LIN {X 0,Y 305.104,Z 484.661,A -85,B 0,C 180,E1 7191.33,E2 7191.33} C_VEL
LIN {X 0,Y 307.303,Z 489.456,A -85,B 0,C 180,E1 7188.457,E2 7188.457} C_VEL
LIN {X 0,Y 307.394,Z 489.963,A -85,B 0,C 180,E1 7188.319,E2 7188.319} C_VEL
LIN {X 0,Y 295.914,Z 597.326,A -85,B 0,C 180,E1 7186.379,E2 7186.379} C_VEL
LIN {X 0,Y 291.472,Z 621.219,A -85,B 0,C 180,E1 7185.834,E2 7185.834} C_VEL
LIN {X 0,Y 286.108,Z 641.71,A -85,B 0,C 180,E1 7185.236,E2 7185.236} C_VEL
LIN {X 0,Y 278.769,Z 663.649,A -85,B 0,C 180,E1 7184.366,E2 7184.366} C_VEL
LIN {X 0,Y 271.258,Z 681.916,A -85,B 0,C 180,E1 7183.403,E2 7183.403} C_VEL
LIN {X 0,Y 262.549,Z 700.2,A -85,B 0,C 180,E1 7182.184,E2 7182.184} C_VEL
LIN {X 0,Y 251.426,Z 720.077,A -85,B 0,C 180,E1 7180.47,E2 7180.47} C_VEL
LIN {X 0,Y 241.401,Z 735.774,A -85,B 0,C 180,E1 7178.733,E2 7178.733} C_VEL
LIN {X 0,Y 229.63,Z 752.334,A -85,B 0,C 180,E1 7176.424,E2 7176.424} C_VEL
LIN {X 0,Y 216.754,Z 768.298,A -85,B 0,C 180,E1 7173.492,E2 7173.492} C_VEL
LIN {X 0,Y 205.612,Z 780.95,A -85,B 0,C 180,E1 7170.508,E2 7170.508} C_VEL
LIN {X 0,Y 192.249,Z 794.919,A -85,B 0,C 180,E1 7166.187,E2 7166.187} C_VEL
LIN {X 0,Y 189.925,Z 797.18,A -85,B 0,C 180,E1 7165.331,E2 7165.331} C_VEL
LIN {X 0,Y 185.106,Z 801.348,A -85,B 0,C 180,E1 7163.939,E2 7163.939} C_VEL
LIN {X 0,Y 170.53,Z 810.999,A -85,B 0,C 180,E1 7160.73,E2 7160.73} C_VEL
LIN {X 0,Y 165.908,Z 814.382,A -85,B 0,C 180,E1 7158.968,E2 7158.968} C_VEL
LIN {X 0,Y 154.577,Z 824.022,A -85,B 0,C 180,E1 7151.776,E2 7151.776} C_VEL
LIN {X 0,Y 146.89,Z 830.6,A -85,B 0,C 180,E1 7144.873,E2 7144.873} C_VEL
LIN {X 0,Y 140.749,Z 836.382,A -85,B 0,C 180,E1 7136.481,E2 7136.481} C_VEL
LIN {X 0,Y 137.18,Z 840.393,A -85,B 0,C 180,E1 7127.387,E2 7127.387} C_VEL
LIN {X 0,Y 136.118,Z 842.389,A -85,B 0,C 180,E1 7120.154,E2 7120.154} C_VEL
LIN {X 0,Y 136.006,Z 843.295,A -85,B 0,C 180,E1 7113.794,E2 7113.794} C_VEL
LIN {X 0,Y 136.026,Z 843.438,A -85,B 0,C 180,E1 7108.315,E2 7108.315} C_VEL
LIN {X 0,Y 136.046,Z 842.73,A -85,B 0,C 180,E1 7101.548,E2 7101.548} C_VEL
LIN {X 0,Y 136.809,Z 840.957,A -85,B 0,C 180,E1 7094.312,E2 7094.312} C_VEL
LIN {X 0,Y 139.161,Z 837.954,A -85,B 0,C 180,E1 7086.724,E2 7086.724} C_VEL
LIN {X 0,Y 143.968,Z 833.277,A -85,B 0,C 180,E1 7078.61,E2 7078.61} C_VEL
LIN {X 0,Y 151.933,Z 826.255,A -85,B 0,C 180,E1 7070.333,E2 7070.333} C_VEL
LIN {X 0,Y 160.416,Z 819.053,A -85,B 0,C 180,E1 7064.212,E2 7064.212} C_VEL
LIN {X 0,Y 171.771,Z 809.365,A -85,B 0,C 180,E1 7058.098,E2 7058.098} C_VEL
LIN {X 0,Y 183.827,Z 798.354,A -85,B 0,C 180,E1 7053.112,E2 7053.112} C_VEL
LIN {X 0,Y 195.767,Z 786.783,A -85,B 0,C 180,E1 7049.151,E2 7049.151} C_VEL
LIN {X 0,Y 210.081,Z 771.62,A -85,B 0,C 180,E1 7045.276,E2 7045.276} C_VEL
LIN {X 0,Y 221.987,Z 757.619,A -85,B 0,C 180,E1 7042.583,E2 7042.583} C_VEL
LIN {X 0,Y 234.35,Z 741.577,A -85,B 0,C 180,E1 7040.181,E2 7040.181} C_VEL
LIN {X 0,Y 246.233,Z 723.952,A -85,B 0,C 180,E1 7038.166,E2 7038.166} C_VEL
LIN {X 0,Y 256.353,Z 706.973,A -85,B 0,C 180,E1 7036.645,E2 7036.645} C_VEL
LIN {X 0,Y 266.872,Z 686.5,A -85,B 0,C 180,E1 7035.225,E2 7035.225} C_VEL
LIN {X 0,Y 274.893,Z 667.932,A -85,B 0,C 180,E1 7034.233,E2 7034.233} C_VEL
LIN {X 0,Y 282.326,Z 647.454,A -85,B 0,C 180,E1 7033.391,E2 7033.391} C_VEL
LIN {X 0,Y 288.635,Z 625.044,A -85,B 0,C 180,E1 7032.726,E2 7032.726} C_VEL
LIN {X 0,Y 293.049,Z 603.912,A -85,B 0,C 180,E1 7032.239,E2 7032.239} C_VEL
LIN {X 0,Y 296.866,Z 573.803,A -85,B 0,C 180,E1 7031.673,E2 7031.673} C_VEL
LIN {X 0,Y 305.233,Z 495.411,A -85,B 0,C 180,E1 7030.284,E2 7030.284} C_VEL
LIN {X 0,Y 303.319,Z 491.087,A -85,B 0,C 180,E1 7027.386,E2 7027.386} C_VEL
LIN {X 0,Y 302.008,Z 487.906,A -85,B 0,C 180,E1 7024.367,E2 7024.367} C_VEL
LIN {X 0,Y 301.205,Z 486.572,A -85,B 0,C 180,E1 7019.81,E2 7019.81} C_VEL
LIN {X 0,Y 302.134,Z 488.028,A -85,B 0,C 180,E1 7014.874,E2 7014.874} C_VEL
LIN {X 0,Y 303.893,Z 492.391,A -85,B 0,C 180,E1 7011.2,E2 7011.2} C_VEL
LIN {X 0,Y 307.885,Z 499.46,A -85,B 0,C 180,E1 7006.478,E2 7006.478} C_VEL
LIN {X 0,Y 312.909,Z 504.765,A -85,B 0,C 180,E1 7002.617,E2 7002.617} C_VEL
LIN {X 0,Y 316.473,Z 507.473,A -85,B 0,C 180,E1 7000.434,E2 7000.434} C_VEL
LIN {X 0,Y 321.483,Z 511.596,A -85,B 0,C 180,E1 6997.315,E2 6997.315} C_VEL
LIN {X 0,Y 325.724,Z 514.379,A -85,B 0,C 180,E1 6994.353,E2 6994.353} C_VEL
LIN {X 0,Y 327.911,Z 515.873,A -85,B 0,C 180,E1 6992.684,E2 6992.684} C_VEL
LIN {X 0,Y 331.07,Z 519.079,A -85,B 0,C 180,E1 6989.912,E2 6989.912} C_VEL
LIN {X 0,Y 334.513,Z 521.924,A -85,B 0,C 180,E1 6986.43,E2 6986.43} C_VEL
LIN {X 0,Y 336.136,Z 523.16,A -85,B 0,C 180,E1 6984.756,E2 6984.756} C_VEL
LIN {X 0,Y 338.877,Z 526.467,A -85,B 0,C 180,E1 6981.703,E2 6981.703} C_VEL
LIN {X 0,Y 342.275,Z 529.188,A -85,B 0,C 180,E1 6978.013,E2 6978.013} C_VEL
LIN {X 0,Y 344.04,Z 530.411,A -85,B 0,C 180,E1 6976.006,E2 6976.006} C_VEL
LIN {X 0,Y 347.045,Z 534.052,A -85,B 0,C 180,E1 6972.232,E2 6972.232} C_VEL
LIN {X 0,Y 349.83,Z 536.292,A -85,B 0,C 180,E1 6968.715,E2 6968.715} C_VEL
LIN {X 0,Y 352.358,Z 537.818,A -85,B 0,C 180,E1 6965.37,E2 6965.37} C_VEL
LIN {X 0,Y 354.546,Z 540.837,A -85,B 0,C 180,E1 6961.913,E2 6961.913} C_VEL
LIN {X 0,Y 356.813,Z 542.935,A -85,B 0,C 180,E1 6958.265,E2 6958.265} C_VEL
LIN {X 0,Y 358.894,Z 544.236,A -85,B 0,C 180,E1 6954.525,E2 6954.525} C_VEL
LIN {X 0,Y 360.791,Z 545.097,A -85,B 0,C 180,E1 6950.776,E2 6950.776} C_VEL
LIN {X 0,Y 361.998,Z 546.95,A -85,B 0,C 180,E1 6947.521,E2 6947.521} C_VEL
LIN {X 0,Y 363.22,Z 548.56,A -85,B 0,C 180,E1 6943.856,E2 6943.856} C_VEL
LIN {X 0,Y 364.051,Z 549.551,A -85,B 0,C 180,E1 6940.443,E2 6940.443} C_VEL
LIN {X 0,Y 364.784,Z 550.154,A -85,B 0,C 180,E1 6936.768,E2 6936.768} C_VEL
LIN {X 0,Y 365.112,Z 550.448,A -85,B 0,C 180,E1 6933.454,E2 6933.454} C_VEL
LIN {X 0,Y 365.309,Z 550.567,A -85,B 0,C 180,E1 6929.843,E2 6929.843} C_VEL
LIN {X 0,Y 365.099,Z 550.448,A -85,B 0,C 180,E1 6926.389,E2 6926.389} C_VEL
LIN {X 0,Y 364.734,Z 550.083,A -85,B 0,C 180,E1 6922.756,E2 6922.756} C_VEL
LIN {X 0,Y 363.978,Z 549.471,A -85,B 0,C 180,E1 6919.234,E2 6919.234} C_VEL
LIN {X 0,Y 363.085,Z 548.4,A -85,B 0,C 180,E1 6915.651,E2 6915.651} C_VEL
LIN {X 0,Y 361.936,Z 546.859,A -85,B 0,C 180,E1 6912.31,E2 6912.31} C_VEL
LIN {X 0,Y 360.733,Z 545.031,A -85,B 0,C 180,E1 6909.051,E2 6909.051} C_VEL
LIN {X 0,Y 358.895,Z 544.236,A -85,B 0,C 180,E1 6905.475,E2 6905.475} C_VEL
LIN {X 0,Y 356.813,Z 542.935,A -85,B 0,C 180,E1 6901.735,E2 6901.735} C_VEL
LIN {X 0,Y 354.546,Z 540.837,A -85,B 0,C 180,E1 6898.087,E2 6898.087} C_VEL
LIN {X 0,Y 352.358,Z 537.819,A -85,B 0,C 180,E1 6894.63,E2 6894.63} C_VEL
LIN {X 0,Y 349.461,Z 536.056,A -85,B 0,C 180,E1 6890.838,E2 6890.838} C_VEL
LIN {X 0,Y 346.883,Z 533.875,A -85,B 0,C 180,E1 6887.552,E2 6887.552} C_VEL
LIN {X 0,Y 343.927,Z 530.256,A -85,B 0,C 180,E1 6883.866,E2 6883.866} C_VEL
LIN {X 0,Y 340.638,Z 528.014,A -85,B 0,C 180,E1 6880.222,E2 6880.222} C_VEL
LIN {X 0,Y 337.257,Z 524.656,A -85,B 0,C 180,E1 6876.471,E2 6876.471} C_VEL
LIN {X 0,Y 335.469,Z 522.476,A -85,B 0,C 180,E1 6874.492,E2 6874.492} C_VEL
LIN {X 0,Y 331.8,Z 519.751,A -85,B 0,C 180,E1 6870.816,E2 6870.816} C_VEL
LIN {X 0,Y 328.541,Z 516.579,A -85,B 0,C 180,E1 6867.849,E2 6867.849} C_VEL
LIN {X 0,Y 326.725,Z 514.885,A -85,B 0,C 180,E1 6866.342,E2 6866.342} C_VEL
LIN {X 0,Y 322.538,Z 512.398,A -85,B 0,C 180,E1 6863.427,E2 6863.427} C_VEL
LIN {X 0,Y 317.626,Z 508.513,A -85,B 0,C 180,E1 6860.259,E2 6860.259} C_VEL
LIN {X 0,Y 314.164,Z 505.643,A -85,B 0,C 180,E1 6858.173,E2 6858.173} C_VEL
LIN {X 0,Y 308.694,Z 500.604,A -85,B 0,C 180,E1 6854.251,E2 6854.251} C_VEL
LIN {X 0,Y 305.593,Z 495.836,A -85,B 0,C 180,E1 6851.13,E2 6851.13} C_VEL
LIN {X 0,Y 303.288,Z 491.023,A -85,B 0,C 180,E1 6847.768,E2 6847.768} C_VEL
LIN {X 0,Y 301.987,Z 487.887,A -85,B 0,C 180,E1 6844.748,E2 6844.748} C_VEL
LIN {X 0,Y 301.205,Z 486.57,A -85,B 0,C 180,E1 6840.19,E2 6840.19} C_VEL
LIN {X 0,Y 302.119,Z 488.008,A -85,B 0,C 180,E1 6835.349,E2 6835.349} C_VEL
LIN {X 0,Y 303.866,Z 492.356,A -85,B 0,C 180,E1 6831.675,E2 6831.675} C_VEL
LIN {X 0,Y 305.234,Z 495.59,A -85,B 0,C 180,E1 6829.692,E2 6829.692} C_VEL
LIN {X 0,Y 294.112,Z 597.19,A -85,B 0,C 180,E1 6827.898,E2 6827.898} C_VEL
LIN {X 0,Y 289.582,Z 621.099,A -85,B 0,C 180,E1 6827.372,E2 6827.372} C_VEL
LIN {X 0,Y 284.203,Z 641.339,A -85,B 0,C 180,E1 6826.808,E2 6826.808} C_VEL
LIN {X 0,Y 276.75,Z 663.292,A -85,B 0,C 180,E1 6825.979,E2 6825.979} C_VEL
LIN {X 0,Y 268.823,Z 682.187,A -85,B 0,C 180,E1 6825.024,E2 6825.024} C_VEL
LIN {X 0,Y 259.301,Z 701.676,A -85,B 0,C 180,E1 6823.762,E2 6823.762} C_VEL
LIN {X 0,Y 248.577,Z 720.215,A -85,B 0,C 180,E1 6822.2,E2 6822.2} C_VEL
LIN {X 0,Y 238.137,Z 736.139,A -85,B 0,C 180,E1 6820.489,E2 6820.489} C_VEL
LIN {X 0,Y 225.247,Z 753.642,A -85,B 0,C 180,E1 6818.081,E2 6818.081} C_VEL
LIN {X 0,Y 212.424,Z 768.939,A -85,B 0,C 180,E1 6815.286,E2 6815.286} C_VEL
LIN {X 0,Y 200.185,Z 782.301,A -85,B 0,C 180,E1 6812.133,E2 6812.133} C_VEL
LIN {X 0,Y 186.553,Z 795.792,A -85,B 0,C 180,E1 6807.865,E2 6807.865} C_VEL
LIN {X 0,Y 175.348,Z 806.096,A -85,B 0,C 180,E1 6803.512,E2 6803.512} C_VEL
LIN {X 0,Y 165.908,Z 814.382,A -85,B 0,C 180,E1 6798.968,E2 6798.968} C_VEL
LIN {X 0,Y 161.388,Z 817.688,A -85,B 0,C 180,E1 6797.08,E2 6797.08} C_VEL
LIN {X 0,Y 147.59,Z 825.211,A -85,B 0,C 180,E1 6792.401,E2 6792.401} C_VEL
LIN {X 0,Y 143.546,Z 827.744,A -85,B 0,C 180,E1 6789.986,E2 6789.986} C_VEL
LIN {X 0,Y 135.713,Z 834.039,A -85,B 0,C 180,E1 6781.539,E2 6781.539} C_VEL
LIN {X 0,Y 131.259,Z 838.095,A -85,B 0,C 180,E1 6773.81,E2 6773.81} C_VEL
LIN {X 0,Y 128.634,Z 841.269,A -85,B 0,C 180,E1 6764.862,E2 6764.862} C_VEL
LIN {X 0,Y 128.003,Z 842.929,A -85,B 0,C 180,E1 6755.828,E2 6755.828} C_VEL
LIN {X 0,Y 128.039,Z 843.245,A -85,B 0,C 180,E1 6749.105,E2 6749.105} C_VEL
LIN {X 0,Y 128.035,Z 842.65,A -85,B 0,C 180,E1 6741.92,E2 6741.92} C_VEL
LIN {X 0,Y 128.976,Z 840.706,A -85,B 0,C 180,E1 6733.332,E2 6733.332} C_VEL
LIN {X 0,Y 131.655,Z 837.701,A -85,B 0,C 180,E1 6725.311,E2 6725.311} C_VEL
LIN {X 0,Y 137.315,Z 832.769,A -85,B 0,C 180,E1 6716.401,E2 6716.401} C_VEL
LIN {X 0,Y 146.11,Z 825.628,A -85,B 0,C 180,E1 6707.886,E2 6707.886} C_VEL
LIN {X 0,Y 155.297,Z 818.363,A -85,B 0,C 180,E1 6701.683,E2 6701.683} C_VEL
LIN {X 0,Y 167.939,Z 808.113,A -85,B 0,C 180,E1 6695.35,E2 6695.35} C_VEL
LIN {X 0,Y 180.145,Z 797.46,A -85,B 0,C 180,E1 6690.653,E2 6690.653} C_VEL
LIN {X 0,Y 192.636,Z 785.812,A -85,B 0,C 180,E1 6686.782,E2 6686.782} C_VEL
LIN {X 0,Y 207.505,Z 770.473,A -85,B 0,C 180,E1 6683.029,E2 6683.029} C_VEL
LIN {X 0,Y 219.801,Z 756.374,A -85,B 0,C 180,E1 6680.438,E2 6680.438} C_VEL
LIN {X 0,Y 232.949,Z 739.582,A -85,B 0,C 180,E1 6678.068,E2 6678.068} C_VEL
LIN {X 0,Y 244.696,Z 722.328,A -85,B 0,C 180,E1 6676.217,E2 6676.217} C_VEL
LIN {X 0,Y 255.803,Z 703.856,A -85,B 0,C 180,E1 6674.676,E2 6674.676} C_VEL
LIN {X 0,Y 265.724,Z 684.378,A -85,B 0,C 180,E1 6673.431,E2 6673.431} C_VEL
LIN {X 0,Y 273.48,Z 666.555,A -85,B 0,C 180,E1 6672.542,E2 6672.542} C_VEL
LIN {X 0,Y 281.084,Z 645.615,A -85,B 0,C 180,E1 6671.741,E2 6671.741} C_VEL
LIN {X 0,Y 287.297,Z 623.474,A -85,B 0,C 180,E1 6671.13,E2 6671.13} C_VEL
LIN {X 0,Y 291.807,Z 601.687,A -85,B 0,C 180,E1 6670.655,E2 6670.655} C_VEL
LIN {X 0,Y 295.891,Z 568.531,A -85,B 0,C 180,E1 6670.06,E2 6670.06} C_VEL
LIN {X 0,Y 303.217,Z 501.505,A -85,B 0,C 180,E1 6668.916,E2 6668.916} C_VEL
LIN {X 0,Y 302.021,Z 498.596,A -85,B 0,C 180,E1 6666.845,E2 6666.845} C_VEL
LIN {X 0,Y 300.963,Z 495.798,A -85,B 0,C 180,E1 6664.191,E2 6664.191} C_VEL
LIN {X 0,Y 300.23,Z 494.512,A -85,B 0,C 180,E1 6659.809,E2 6659.809} C_VEL
LIN {X 0,Y 301.08,Z 495.958,A -85,B 0,C 180,E1 6655.047,E2 6655.047} C_VEL
LIN {X 0,Y 302.72,Z 500.238,A -85,B 0,C 180,E1 6651.452,E2 6651.452} C_VEL
LIN {X 0,Y 306.511,Z 507.154,A -85,B 0,C 180,E1 6646.8,E2 6646.8} C_VEL
LIN {X 0,Y 311.554,Z 512.565,A -85,B 0,C 180,E1 6642.827,E2 6642.827} C_VEL
LIN {X 0,Y 315.236,Z 515.434,A -85,B 0,C 180,E1 6640.547,E2 6640.547} C_VEL
LIN {X 0,Y 320.279,Z 519.511,A -85,B 0,C 180,E1 6637.419,E2 6637.419} C_VEL
LIN {X 0,Y 324.569,Z 522.278,A -85,B 0,C 180,E1 6634.451,E2 6634.451} C_VEL
LIN {X 0,Y 326.675,Z 523.725,A -85,B 0,C 180,E1 6632.868,E2 6632.868} C_VEL
LIN {X 0,Y 329.974,Z 527.007,A -85,B 0,C 180,E1 6630.002,E2 6630.002} C_VEL
LIN {X 0,Y 333.437,Z 529.838,A -85,B 0,C 180,E1 6626.513,E2 6626.513} C_VEL
LIN {X 0,Y 335.057,Z 531.131,A -85,B 0,C 180,E1 6624.849,E2 6624.849} C_VEL
LIN {X 0,Y 337.987,Z 534.563,A -85,B 0,C 180,E1 6621.594,E2 6621.594} C_VEL
LIN {X 0,Y 341.397,Z 537.221,A -85,B 0,C 180,E1 6617.881,E2 6617.881} C_VEL
LIN {X 0,Y 342.997,Z 538.414,A -85,B 0,C 180,E1 6616.055,E2 6616.055} C_VEL
LIN {X 0,Y 346.014,Z 541.999,A -85,B 0,C 180,E1 6612.29,E2 6612.29} C_VEL
LIN {X 0,Y 348.889,Z 544.276,A -85,B 0,C 180,E1 6608.663,E2 6608.663} C_VEL
LIN {X 0,Y 351.365,Z 545.841,A -85,B 0,C 180,E1 6605.373,E2 6605.373} C_VEL
LIN {X 0,Y 353.555,Z 548.808,A -85,B 0,C 180,E1 6601.926,E2 6601.926} C_VEL
LIN {X 0,Y 355.893,Z 550.929,A -85,B 0,C 180,E1 6598.162,E2 6598.162} C_VEL
LIN {X 0,Y 357.98,Z 552.213,A -85,B 0,C 180,E1 6594.416,E2 6594.416} C_VEL
LIN {X 0,Y 359.918,Z 553.152,A -85,B 0,C 180,E1 6590.489,E2 6590.489} C_VEL
LIN {X 0,Y 361.2,Z 555.135,A -85,B 0,C 180,E1 6587.063,E2 6587.063} C_VEL
LIN {X 0,Y 362.335,Z 556.681,A -85,B 0,C 180,E1 6583.403,E2 6583.403} C_VEL
LIN {X 0,Y 363.152,Z 557.557,A -85,B 0,C 180,E1 6580.149,E2 6580.149} C_VEL
LIN {X 0,Y 363.837,Z 558.169,A -85,B 0,C 180,E1 6576.311,E2 6576.311} C_VEL
LIN {X 0,Y 364.171,Z 558.392,A -85,B 0,C 180,E1 6573.148,E2 6573.148} C_VEL
LIN {X 0,Y 364.271,Z 558.474,A -85,B 0,C 180,E1 6569.214,E2 6569.214} C_VEL
LIN {X 0,Y 364.104,Z 558.382,A -85,B 0,C 180,E1 6566.064,E2 6566.064} C_VEL
LIN {X 0,Y 363.626,Z 557.966,A -85,B 0,C 180,E1 6562.257,E2 6562.257} C_VEL
LIN {X 0,Y 362.964,Z 557.365,A -85,B 0,C 180,E1 6559.043,E2 6559.043} C_VEL
LIN {X 0,Y 361.931,Z 556.198,A -85,B 0,C 180,E1 6555.216,E2 6555.216} C_VEL
LIN {X 0,Y 360.821,Z 554.591,A -85,B 0,C 180,E1 6551.892,E2 6551.892} C_VEL
LIN {X 0,Y 359.66,Z 552.924,A -85,B 0,C 180,E1 6548.814,E2 6548.814} C_VEL
LIN {X 0,Y 357.774,Z 552.107,A -85,B 0,C 180,E1 6545.217,E2 6545.217} C_VEL
LIN {X 0,Y 355.654,Z 550.764,A -85,B 0,C 180,E1 6541.451,E2 6541.451} C_VEL
LIN {X 0,Y 353.372,Z 548.597,A -85,B 0,C 180,E1 6537.78,E2 6537.78} C_VEL
LIN {X 0,Y 350.934,Z 545.355,A -85,B 0,C 180,E1 6534.013,E2 6534.013} C_VEL
LIN {X 0,Y 348.262,Z 543.866,A -85,B 0,C 180,E1 6530.561,E2 6530.561} C_VEL
LIN {X 0,Y 345.413,Z 541.344,A -85,B 0,C 180,E1 6526.912,E2 6526.912} C_VEL
LIN {X 0,Y 342.236,Z 537.7,A -85,B 0,C 180,E1 6523.083,E2 6523.083} C_VEL
LIN {X 0,Y 338.9,Z 535.355,A -85,B 0,C 180,E1 6519.369,E2 6519.369} C_VEL
LIN {X 0,Y 335.707,Z 532.044,A -85,B 0,C 180,E1 6515.895,E2 6515.895} C_VEL
LIN {X 0,Y 334.207,Z 530.288,A -85,B 0,C 180,E1 6514.225,E2 6514.225} C_VEL
LIN {X 0,Y 330.693,Z 527.675,A -85,B 0,C 180,E1 6510.729,E2 6510.729} C_VEL
LIN {X 0,Y 327.403,Z 524.538,A -85,B 0,C 180,E1 6507.757,E2 6507.757} C_VEL
LIN {X 0,Y 325.563,Z 522.782,A -85,B 0,C 180,E1 6506.247,E2 6506.247} C_VEL
LIN {X 0,Y 321.293,Z 520.261,A -85,B 0,C 180,E1 6503.28,E2 6503.28} C_VEL
LIN {X 0,Y 316.092,Z 516.207,A -85,B 0,C 180,E1 6499.976,E2 6499.976} C_VEL
LIN {X 0,Y 312.652,Z 513.348,A -85,B 0,C 180,E1 6497.879,E2 6497.879} C_VEL
LIN {X 0,Y 307.197,Z 508.156,A -85,B 0,C 180,E1 6493.841,E2 6493.841} C_VEL
LIN {X 0,Y 304.217,Z 503.402,A -85,B 0,C 180,E1 6490.702,E2 6490.702} C_VEL
LIN {X 0,Y 302.093,Z 498.728,A -85,B 0,C 180,E1 6487.416,E2 6487.416} C_VEL
LIN {X 0,Y 300.944,Z 495.778,A -85,B 0,C 180,E1 6484.573,E2 6484.573} C_VEL
LIN {X 0,Y 300.23,Z 494.511,A -85,B 0,C 180,E1 6480.191,E2 6480.191} C_VEL
LIN {X 0,Y 301.069,Z 495.911,A -85,B 0,C 180,E1 6475.524,E2 6475.524} C_VEL
LIN {X 0,Y 302.693,Z 500.201,A -85,B 0,C 180,E1 6471.93,E2 6471.93} C_VEL
LIN {X 0,Y 303.193,Z 501.752,A -85,B 0,C 180,E1 6471.075,E2 6471.075} C_VEL
LIN {X 0,Y 292.52,Z 597.054,A -85,B 0,C 180,E1 6469.435,E2 6469.435} C_VEL
LIN {X 0,Y 287.904,Z 620.979,A -85,B 0,C 180,E1 6468.929,E2 6468.929} C_VEL
LIN {X 0,Y 282.244,Z 641.883,A -85,B 0,C 180,E1 6468.373,E2 6468.373} C_VEL
LIN {X 0,Y 274.4,Z 664.292,A -85,B 0,C 180,E1 6467.557,E2 6467.557} C_VEL
LIN {X 0,Y 266.55,Z 682.583,A -85,B 0,C 180,E1 6466.668,E2 6466.668} C_VEL
LIN {X 0,Y 256.582,Z 702.448,A -85,B 0,C 180,E1 6465.425,E2 6465.425} C_VEL
LIN {X 0,Y 245.576,Z 720.953,A -85,B 0,C 180,E1 6463.913,E2 6463.913} C_VEL
LIN {X 0,Y 235.102,Z 736.504,A -85,B 0,C 180,E1 6462.291,E2 6462.291} C_VEL
LIN {X 0,Y 222.007,Z 753.757,A -85,B 0,C 180,E1 6459.984,E2 6459.984} C_VEL
LIN {X 0,Y 209.119,Z 768.686,A -85,B 0,C 180,E1 6457.334,E2 6457.334} C_VEL
LIN {X 0,Y 196.465,Z 782.047,A -85,B 0,C 180,E1 6454.26,E2 6454.26} C_VEL
LIN {X 0,Y 182.205,Z 795.61,A -85,B 0,C 180,E1 6450.042,E2 6450.042} C_VEL
LIN {X 0,Y 170.54,Z 805.849,A -85,B 0,C 180,E1 6445.748,E2 6445.748} C_VEL
LIN {X 0,Y 158.134,Z 816.181,A -85,B 0,C 180,E1 6439.911,E2 6439.911} C_VEL
LIN {X 0,Y 147.526,Z 824.512,A -85,B 0,C 180,E1 6433.197,E2 6433.197} C_VEL
LIN {X 0,Y 143.546,Z 827.744,A -85,B 0,C 180,E1 6429.986,E2 6429.986} C_VEL
LIN {X 0,Y 139.719,Z 830.079,A -85,B 0,C 180,E1 6427.42,E2 6427.42} C_VEL
LIN {X 0,Y 127.339,Z 835.519,A -85,B 0,C 180,E1 6420.361,E2 6420.361} C_VEL
LIN {X 0,Y 124.923,Z 836.877,A -85,B 0,C 180,E1 6417.603,E2 6417.603} C_VEL
LIN {X 0,Y 121.418,Z 840.172,A -85,B 0,C 180,E1 6408.732,E2 6408.732} C_VEL
LIN {X 0,Y 120.14,Z 842.06,A -85,B 0,C 180,E1 6400.55,E2 6400.55} C_VEL
LIN {X 0,Y 120.011,Z 842.828,A -85,B 0,C 180,E1 6393.822,E2 6393.822} C_VEL
LIN {X 0,Y 120.03,Z 842.942,A -85,B 0,C 180,E1 6388.091,E2 6388.091} C_VEL
LIN {X 0,Y 120.067,Z 842.316,A -85,B 0,C 180,E1 6380.896,E2 6380.896} C_VEL
LIN {X 0,Y 121.181,Z 840.455,A -85,B 0,C 180,E1 6372.225,E2 6372.225} C_VEL
LIN {X 0,Y 124.234,Z 837.448,A -85,B 0,C 180,E1 6363.728,E2 6363.728} C_VEL
LIN {X 0,Y 130.508,Z 832.515,A -85,B 0,C 180,E1 6354.392,E2 6354.392} C_VEL
LIN {X 0,Y 140.071,Z 825.373,A -85,B 0,C 180,E1 6345.611,E2 6345.611} C_VEL
LIN {X 0,Y 149.906,Z 818.107,A -85,B 0,C 180,E1 6339.314,E2 6339.314} C_VEL
LIN {X 0,Y 163.283,Z 807.854,A -85,B 0,C 180,E1 6332.977,E2 6332.977} C_VEL
LIN {X 0,Y 176.068,Z 797.206,A -85,B 0,C 180,E1 6328.335,E2 6328.335} C_VEL
LIN {X 0,Y 189.848,Z 784.84,A -85,B 0,C 180,E1 6324.342,E2 6324.342} C_VEL
LIN {X 0,Y 204.427,Z 770.22,A -85,B 0,C 180,E1 6320.907,E2 6320.907} C_VEL
LIN {X 0,Y 217.073,Z 756.123,A -85,B 0,C 180,E1 6318.409,E2 6318.409} C_VEL
LIN {X 0,Y 230.806,Z 738.968,A -85,B 0,C 180,E1 6316.096,E2 6316.096} C_VEL
LIN {X 0,Y 242.547,Z 722.078,A -85,B 0,C 180,E1 6314.369,E2 6314.369} C_VEL
LIN {X 0,Y 253.869,Z 703.601,A -85,B 0,C 180,E1 6312.904,E2 6312.904} C_VEL
LIN {X 0,Y 263.962,Z 684.13,A -85,B 0,C 180,E1 6311.723,E2 6311.723} C_VEL
LIN {X 0,Y 271.843,Z 666.311,A -85,B 0,C 180,E1 6310.882,E2 6310.882} C_VEL
LIN {X 0,Y 279.582,Z 645.287,A -85,B 0,C 180,E1 6310.124,E2 6310.124} C_VEL
LIN {X 0,Y 285.87,Z 623.176,A -85,B 0,C 180,E1 6309.549,E2 6309.549} C_VEL
LIN {X 0,Y 290.461,Z 601.249,A -85,B 0,C 180,E1 6309.093,E2 6309.093} C_VEL
LIN {X 0,Y 294.664,Z 567.644,A -85,B 0,C 180,E1 6308.511,E2 6308.511} C_VEL
LIN {X 0,Y 301.352,Z 507.516,A -85,B 0,C 180,E1 6307.483,E2 6307.483} C_VEL
LIN {X 0,Y 299.922,Z 503.689,A -85,B 0,C 180,E1 6304.014,E2 6304.014} C_VEL
LIN {X 0,Y 299.256,Z 502.456,A -85,B 0,C 180,E1 6299.617,E2 6299.617} C_VEL
LIN {X 0,Y 300.055,Z 504.002,A -85,B 0,C 180,E1 6295.126,E2 6295.126} C_VEL
LIN {X 0,Y 301.502,Z 507.934,A -85,B 0,C 180,E1 6291.802,E2 6291.802} C_VEL
LIN {X 0,Y 305.522,Z 515.426,A -85,B 0,C 180,E1 6286.757,E2 6286.757} C_VEL
LIN {X 0,Y 310.604,Z 520.663,A -85,B 0,C 180,E1 6282.773,E2 6282.773} C_VEL
LIN {X 0,Y 314.002,Z 523.39,A -85,B 0,C 180,E1 6280.661,E2 6280.661} C_VEL
LIN {X 0,Y 319.064,Z 527.423,A -85,B 0,C 180,E1 6277.523,E2 6277.523} C_VEL
LIN {X 0,Y 323.505,Z 530.225,A -85,B 0,C 180,E1 6274.483,E2 6274.483} C_VEL
LIN {X 0,Y 325.554,Z 531.707,A -85,B 0,C 180,E1 6272.954,E2 6272.954} C_VEL
LIN {X 0,Y 329.054,Z 535.105,A -85,B 0,C 180,E1 6269.91,E2 6269.91} C_VEL
LIN {X 0,Y 332.551,Z 537.87,A -85,B 0,C 180,E1 6266.412,E2 6266.412} C_VEL
LIN {X 0,Y 333.917,Z 539.012,A -85,B 0,C 180,E1 6265.011,E2 6265.011} C_VEL
LIN {X 0,Y 336.926,Z 542.498,A -85,B 0,C 180,E1 6261.668,E2 6261.668} C_VEL
LIN {X 0,Y 340.35,Z 545.143,A -85,B 0,C 180,E1 6257.948,E2 6257.948} C_VEL
LIN {X 0,Y 341.819,Z 546.232,A -85,B 0,C 180,E1 6256.26,E2 6256.26} C_VEL
LIN {X 0,Y 344.863,Z 549.826,A -85,B 0,C 180,E1 6252.494,E2 6252.494} C_VEL
LIN {X 0,Y 347.591,Z 552.036,A -85,B 0,C 180,E1 6249.044,E2 6249.044} C_VEL
LIN {X 0,Y 350.271,Z 553.685,A -85,B 0,C 180,E1 6245.557,E2 6245.557} C_VEL
LIN {X 0,Y 352.525,Z 556.735,A -85,B 0,C 180,E1 6242,E2 6242} C_VEL
LIN {X 0,Y 354.74,Z 558.767,A -85,B 0,C 180,E1 6238.431,E2 6238.431} C_VEL
LIN {X 0,Y 356.857,Z 560.083,A -85,B 0,C 180,E1 6234.675,E2 6234.675} C_VEL
LIN {X 0,Y 358.797,Z 560.954,A -85,B 0,C 180,E1 6230.897,E2 6230.897} C_VEL
LIN {X 0,Y 360.065,Z 562.906,A -85,B 0,C 180,E1 6227.451,E2 6227.451} C_VEL
LIN {X 0,Y 361.287,Z 564.507,A -85,B 0,C 180,E1 6223.739,E2 6223.739} C_VEL
LIN {X 0,Y 362.126,Z 565.462,A -85,B 0,C 180,E1 6220.339,E2 6220.339} C_VEL
LIN {X 0,Y 362.838,Z 566.06,A -85,B 0,C 180,E1 6216.646,E2 6216.646} C_VEL
LIN {X 0,Y 363.177,Z 566.33,A -85,B 0,C 180,E1 6213.314,E2 6213.314} C_VEL
LIN {X 0,Y 363.339,Z 566.44,A -85,B 0,C 180,E1 6209.685,E2 6209.685} C_VEL
LIN {X 0,Y 363.148,Z 566.328,A -85,B 0,C 180,E1 6206.369,E2 6206.369} C_VEL
LIN {X 0,Y 362.799,Z 565.974,A -85,B 0,C 180,E1 6202.812,E2 6202.812} C_VEL
LIN {X 0,Y 362.049,Z 565.388,A -85,B 0,C 180,E1 6199.337,E2 6199.337} C_VEL
LIN {X 0,Y 361.148,Z 564.309,A -85,B 0,C 180,E1 6195.694,E2 6195.694} C_VEL
LIN {X 0,Y 359.943,Z 562.732,A -85,B 0,C 180,E1 6192.209,E2 6192.209} C_VEL
LIN {X 0,Y 358.738,Z 560.892,A -85,B 0,C 180,E1 6188.928,E2 6188.928} C_VEL
LIN {X 0,Y 356.801,Z 560.053,A -85,B 0,C 180,E1 6185.222,E2 6185.222} C_VEL
LIN {X 0,Y 354.731,Z 558.761,A -85,B 0,C 180,E1 6181.554,E2 6181.554} C_VEL
LIN {X 0,Y 352.505,Z 556.713,A -85,B 0,C 180,E1 6177.968,E2 6177.968} C_VEL
LIN {X 0,Y 350.233,Z 553.626,A -85,B 0,C 180,E1 6174.383,E2 6174.383} C_VEL
LIN {X 0,Y 347.238,Z 551.797,A -85,B 0,C 180,E1 6170.506,E2 6170.506} C_VEL
LIN {X 0,Y 344.487,Z 549.408,A -85,B 0,C 180,E1 6166.995,E2 6166.995} C_VEL
LIN {X 0,Y 341.578,Z 545.894,A -85,B 0,C 180,E1 6163.455,E2 6163.455} C_VEL
LIN {X 0,Y 338.296,Z 543.659,A -85,B 0,C 180,E1 6159.787,E2 6159.787} C_VEL
LIN {X 0,Y 334.925,Z 540.369,A -85,B 0,C 180,E1 6156.129,E2 6156.129} C_VEL
LIN {X 0,Y 333.026,Z 538.142,A -85,B 0,C 180,E1 6154.042,E2 6154.042} C_VEL
LIN {X 0,Y 329.588,Z 535.598,A -85,B 0,C 180,E1 6150.641,E2 6150.641} C_VEL
LIN {X 0,Y 326.281,Z 532.509,A -85,B 0,C 180,E1 6147.676,E2 6147.676} C_VEL
LIN {X 0,Y 324.15,Z 530.557,A -85,B 0,C 180,E1 6145.977,E2 6145.977} C_VEL
LIN {X 0,Y 319.865,Z 527.99,A -85,B 0,C 180,E1 6143,E2 6143} C_VEL
LIN {X 0,Y 314.566,Z 523.9,A -85,B 0,C 180,E1 6139.69,E2 6139.69} C_VEL
LIN {X 0,Y 311.15,Z 521.052,A -85,B 0,C 180,E1 6137.581,E2 6137.581} C_VEL
LIN {X 0,Y 305.814,Z 515.847,A -85,B 0,C 180,E1 6133.519,E2 6133.519} C_VEL
LIN {X 0,Y 302.786,Z 510.841,A -85,B 0,C 180,E1 6130.176,E2 6130.176} C_VEL
LIN {X 0,Y 300.911,Z 506.432,A -85,B 0,C 180,E1 6127.062,E2 6127.062} C_VEL
LIN {X 0,Y 299.903,Z 503.669,A -85,B 0,C 180,E1 6124.398,E2 6124.398} C_VEL
LIN {X 0,Y 299.258,Z 502.448,A -85,B 0,C 180,E1 6120,E2 6120} C_VEL
LIN {X 0,Y 300.07,Z 504.069,A -85,B 0,C 180,E1 6115.509,E2 6115.509} C_VEL
LIN {X 0,Y 301.365,Z 507.617,A -85,B 0,C 180,E1 6112.482,E2 6112.482} C_VEL
LIN {X 0,Y 291.139,Z 596.913,A -85,B 0,C 180,E1 6110.987,E2 6110.987} C_VEL
LIN {X 0,Y 286.47,Z 620.74,A -85,B 0,C 180,E1 6110.506,E2 6110.506} C_VEL
LIN {X 0,Y 280.499,Z 642.424,A -85,B 0,C 180,E1 6109.959,E2 6109.959} C_VEL
LIN {X 0,Y 272.776,Z 664.047,A -85,B 0,C 180,E1 6109.211,E2 6109.211} C_VEL
LIN {X 0,Y 264.884,Z 682.158,A -85,B 0,C 180,E1 6108.38,E2 6108.38} C_VEL
LIN {X 0,Y 255.239,Z 701.166,A -85,B 0,C 180,E1 6107.263,E2 6107.263} C_VEL
LIN {X 0,Y 243.895,Z 720.017,A -85,B 0,C 180,E1 6105.816,E2 6105.816} C_VEL
LIN {X 0,Y 232.747,Z 736.253,A -85,B 0,C 180,E1 6104.208,E2 6104.208} C_VEL
LIN {X 0,Y 218.791,Z 754.135,A -85,B 0,C 180,E1 6101.9,E2 6101.9} C_VEL
LIN {X 0,Y 206.09,Z 768.433,A -85,B 0,C 180,E1 6099.444,E2 6099.444} C_VEL
LIN {X 0,Y 192.23,Z 782.596,A -85,B 0,C 180,E1 6096.265,E2 6096.265} C_VEL
LIN {X 0,Y 177.518,Z 795.956,A -85,B 0,C 180,E1 6092.128,E2 6092.128} C_VEL
LIN {X 0,Y 164.647,Z 806.722,A -85,B 0,C 180,E1 6087.574,E2 6087.574} C_VEL
LIN {X 0,Y 150.5,Z 817.672,A -85,B 0,C 180,E1 6081.012,E2 6081.012} C_VEL
LIN {X 0,Y 140.27,Z 825.225,A -85,B 0,C 180,E1 6074.536,E2 6074.536} C_VEL
LIN {X 0,Y 130.679,Z 832.393,A -85,B 0,C 180,E1 6065.803,E2 6065.803} C_VEL
LIN {X 0,Y 124.923,Z 836.877,A -85,B 0,C 180,E1 6057.603,E2 6057.603} C_VEL
LIN {X 0,Y 122.308,Z 838.359,A -85,B 0,C 180,E1 6054.279,E2 6054.279} C_VEL
LIN {X 0,Y 115.553,Z 840.537,A -85,B 0,C 180,E1 6047.836,E2 6047.836} C_VEL
LIN {X 0,Y 112.498,Z 841.535,A -85,B 0,C 180,E1 6043.035,E2 6043.035} C_VEL
LIN {X 0,Y 112.215,Z 841.758,A -85,B 0,C 180,E1 6041.623,E2 6041.623} C_VEL
LIN {X 0,Y 112.012,Z 842.58,A -85,B 0,C 180,E1 6034.095,E2 6034.095} C_VEL
LIN {X 0,Y 112.031,Z 842.694,A -85,B 0,C 180,E1 6027.954,E2 6027.954} C_VEL
LIN {X 0,Y 112.092,Z 842.066,A -85,B 0,C 180,E1 6020.243,E2 6020.243} C_VEL
LIN {X 0,Y 113.433,Z 840.203,A -85,B 0,C 180,E1 6010.966,E2 6010.966} C_VEL
LIN {X 0,Y 117.174,Z 836.998,A -85,B 0,C 180,E1 6001.456,E2 6001.456} C_VEL
LIN {X 0,Y 124.697,Z 831.701,A -85,B 0,C 180,E1 5991.288,E2 5991.288} C_VEL
LIN {X 0,Y 134.813,Z 824.746,A -85,B 0,C 180,E1 5982.758,E2 5982.758} C_VEL
LIN {X 0,Y 146.326,Z 816.802,A -85,B 0,C 180,E1 5975.99,E2 5975.99} C_VEL
LIN {X 0,Y 161.075,Z 805.899,A -85,B 0,C 180,E1 5969.656,E2 5969.656} C_VEL
LIN {X 0,Y 174.621,Z 795.031,A -85,B 0,C 180,E1 5965.222,E2 5965.222} C_VEL
LIN {X 0,Y 189.885,Z 781.54,A -85,B 0,C 180,E1 5961.254,E2 5961.254} C_VEL
LIN {X 0,Y 203.348,Z 768.18,A -85,B 0,C 180,E1 5958.387,E2 5958.387} C_VEL
LIN {X 0,Y 217.266,Z 752.88,A -85,B 0,C 180,E1 5955.889,E2 5955.889} C_VEL
LIN {X 0,Y 231.214,Z 735.242,A -85,B 0,C 180,E1 5953.759,E2 5953.759} C_VEL
LIN {X 0,Y 242.488,Z 719.08,A -85,B 0,C 180,E1 5952.258,E2 5952.258} C_VEL
LIN {X 0,Y 254.501,Z 699.214,A -85,B 0,C 180,E1 5950.843,E2 5950.843} C_VEL
LIN {X 0,Y 263.843,Z 680.923,A -85,B 0,C 180,E1 5949.847,E2 5949.847} C_VEL
LIN {X 0,Y 272.33,Z 661.528,A -85,B 0,C 180,E1 5949.03,E2 5949.03} C_VEL
LIN {X 0,Y 279.923,Z 639.837,A -85,B 0,C 180,E1 5948.354,E2 5948.354} C_VEL
LIN {X 0,Y 285.774,Z 618.42,A -85,B 0,C 180,E1 5947.86,E2 5947.86} C_VEL
LIN {X 0,Y 290.222,Z 594.937,A -85,B 0,C 180,E1 5947.415,E2 5947.415} C_VEL
LIN {X 0,Y 299.655,Z 513.953,A -85,B 0,C 180,E1 5946.086,E2 5946.086} C_VEL
LIN {X 0,Y 298.822,Z 511.51,A -85,B 0,C 180,E1 5943.645,E2 5943.645} C_VEL
LIN {X 0,Y 298.281,Z 510.396,A -85,B 0,C 180,E1 5939.616,E2 5939.616} C_VEL
LIN {X 0,Y 298.982,Z 511.809,A -85,B 0,C 180,E1 5935.396,E2 5935.396} C_VEL
LIN {X 0,Y 300.294,Z 515.629,A -85,B 0,C 180,E1 5932.154,E2 5932.154} C_VEL
LIN {X 0,Y 304.345,Z 523.399,A -85,B 0,C 180,E1 5926.898,E2 5926.898} C_VEL
LIN {X 0,Y 309.655,Z 528.756,A -85,B 0,C 180,E1 5922.719,E2 5922.719} C_VEL
LIN {X 0,Y 316.598,Z 534.427,A -85,B 0,C 180,E1 5918.413,E2 5918.413} C_VEL
LIN {X 0,Y 321.006,Z 537.381,A -85,B 0,C 180,E1 5915.527,E2 5915.527} C_VEL
LIN {X 0,Y 324.042,Z 539.301,A -85,B 0,C 180,E1 5913.324,E2 5913.324} C_VEL
LIN {X 0,Y 327.751,Z 542.86,A -85,B 0,C 180,E1 5910.181,E2 5910.181} C_VEL
LIN {X 0,Y 331.236,Z 545.634,A -85,B 0,C 180,E1 5906.733,E2 5906.733} C_VEL
LIN {X 0,Y 332.759,Z 546.877,A -85,B 0,C 180,E1 5905.187,E2 5905.187} C_VEL
LIN {X 0,Y 335.866,Z 550.433,A -85,B 0,C 180,E1 5901.742,E2 5901.742} C_VEL
LIN {X 0,Y 339.302,Z 553.065,A -85,B 0,C 180,E1 5898.016,E2 5898.016} C_VEL
LIN {X 0,Y 340.79,Z 554.246,A -85,B 0,C 180,E1 5896.295,E2 5896.295} C_VEL
LIN {X 0,Y 343.775,Z 557.715,A -85,B 0,C 180,E1 5892.622,E2 5892.622} C_VEL
LIN {X 0,Y 346.565,Z 559.966,A -85,B 0,C 180,E1 5889.097,E2 5889.097} C_VEL
LIN {X 0,Y 349.248,Z 561.661,A -85,B 0,C 180,E1 5885.604,E2 5885.604} C_VEL
LIN {X 0,Y 351.515,Z 564.683,A -85,B 0,C 180,E1 5882.045,E2 5882.045} C_VEL
LIN {X 0,Y 353.809,Z 566.755,A -85,B 0,C 180,E1 5878.343,E2 5878.343} C_VEL
LIN {X 0,Y 355.983,Z 568.081,A -85,B 0,C 180,E1 5874.491,E2 5874.491} C_VEL
LIN {X 0,Y 357.921,Z 569.009,A -85,B 0,C 180,E1 5870.608,E2 5870.608} C_VEL
LIN {X 0,Y 359.2,Z 571.004,A -85,B 0,C 180,E1 5867.161,E2 5867.161} C_VEL
LIN {X 0,Y 360.401,Z 572.616,A -85,B 0,C 180,E1 5863.312,E2 5863.312} C_VEL
LIN {X 0,Y 361.233,Z 573.457,A -85,B 0,C 180,E1 5860.042,E2 5860.042} C_VEL
LIN {X 0,Y 361.883,Z 574.048,A -85,B 0,C 180,E1 5856.345,E2 5856.345} C_VEL
LIN {X 0,Y 362.22,Z 574.273,A -85,B 0,C 180,E1 5853.165,E2 5853.165} C_VEL
LIN {X 0,Y 362.333,Z 574.362,A -85,B 0,C 180,E1 5849.368,E2 5849.368} C_VEL
LIN {X 0,Y 362.161,Z 574.266,A -85,B 0,C 180,E1 5846.201,E2 5846.201} C_VEL
LIN {X 0,Y 361.747,Z 573.874,A -85,B 0,C 180,E1 5842.536,E2 5842.536} C_VEL
LIN {X 0,Y 361.031,Z 573.285,A -85,B 0,C 180,E1 5839.145,E2 5839.145} C_VEL
LIN {X 0,Y 360.032,Z 572.147,A -85,B 0,C 180,E1 5835.362,E2 5835.362} C_VEL
LIN {X 0,Y 358.892,Z 570.578,A -85,B 0,C 180,E1 5831.987,E2 5831.987} C_VEL
LIN {X 0,Y 357.729,Z 568.821,A -85,B 0,C 180,E1 5828.866,E2 5828.866} C_VEL
LIN {X 0,Y 355.805,Z 567.988,A -85,B 0,C 180,E1 5825.185,E2 5825.185} C_VEL
LIN {X 0,Y 353.692,Z 566.673,A -85,B 0,C 180,E1 5821.462,E2 5821.462} C_VEL
LIN {X 0,Y 351.332,Z 564.472,A -85,B 0,C 180,E1 5817.655,E2 5817.655} C_VEL
LIN {X 0,Y 348.697,Z 561.133,A -85,B 0,C 180,E1 5813.682,E2 5813.682} C_VEL
LIN {X 0,Y 345.948,Z 559.532,A -85,B 0,C 180,E1 5810.088,E2 5810.088} C_VEL
LIN {X 0,Y 342.899,Z 556.827,A -85,B 0,C 180,E1 5806.314,E2 5806.314} C_VEL
LIN {X 0,Y 340.014,Z 553.47,A -85,B 0,C 180,E1 5802.788,E2 5802.788} C_VEL
LIN {X 0,Y 336.413,Z 550.911,A -85,B 0,C 180,E1 5798.838,E2 5798.838} C_VEL
LIN {X 0,Y 333.252,Z 547.572,A -85,B 0,C 180,E1 5795.384,E2 5795.384} C_VEL
LIN {X 0,Y 331.86,Z 546.008,A -85,B 0,C 180,E1 5793.875,E2 5793.875} C_VEL
LIN {X 0,Y 328.46,Z 543.494,A -85,B 0,C 180,E1 5790.52,E2 5790.52} C_VEL
LIN {X 0,Y 324.921,Z 540.226,A -85,B 0,C 180,E1 5787.39,E2 5787.39} C_VEL
LIN {X 0,Y 322.744,Z 538.33,A -85,B 0,C 180,E1 5785.704,E2 5785.704} C_VEL
LIN {X 0,Y 318.395,Z 535.713,A -85,B 0,C 180,E1 5782.722,E2 5782.722} C_VEL
LIN {X 0,Y 313.189,Z 531.718,A -85,B 0,C 180,E1 5779.488,E2 5779.488} C_VEL
LIN {X 0,Y 309.386,Z 528.562,A -85,B 0,C 180,E1 5777.103,E2 5777.103} C_VEL
LIN {X 0,Y 304.157,Z 523.118,A -85,B 0,C 180,E1 5772.917,E2 5772.917} C_VEL
LIN {X 0,Y 301.449,Z 518.403,A -85,B 0,C 180,E1 5769.739,E2 5769.739} C_VEL
LIN {X 0,Y 299.739,Z 514.135,A -85,B 0,C 180,E1 5766.705,E2 5766.705} C_VEL
LIN {X 0,Y 298.866,Z 511.559,A -85,B 0,C 180,E1 5764.221,E2 5764.221} C_VEL
LIN {X 0,Y 298.283,Z 510.389,A -85,B 0,C 180,E1 5760,E2 5760} C_VEL
LIN {X 0,Y 298.995,Z 511.874,A -85,B 0,C 180,E1 5755.781,E2 5755.781} C_VEL
LIN {X 0,Y 299.649,Z 514.096,A -85,B 0,C 180,E1 5753.894,E2 5753.894} C_VEL
LIN {X 0,Y 289.96,Z 596.862,A -85,B 0,C 180,E1 5752.552,E2 5752.552} C_VEL
LIN {X 0,Y 285.225,Z 620.62,A -85,B 0,C 180,E1 5752.095,E2 5752.095} C_VEL
LIN {X 0,Y 279.209,Z 642.184,A -85,B 0,C 180,E1 5751.584,E2 5751.584} C_VEL
LIN {X 0,Y 271.382,Z 663.803,A -85,B 0,C 180,E1 5750.884,E2 5750.884} C_VEL
LIN {X 0,Y 263.374,Z 681.909,A -85,B 0,C 180,E1 5750.105,E2 5750.105} C_VEL
LIN {X 0,Y 253.109,Z 701.722,A -85,B 0,C 180,E1 5748.999,E2 5748.999} C_VEL
LIN {X 0,Y 241.571,Z 720.455,A -85,B 0,C 180,E1 5747.627,E2 5747.627} C_VEL
LIN {X 0,Y 230.207,Z 736.618,A -85,B 0,C 180,E1 5746.096,E2 5746.096} C_VEL
LIN {X 0,Y 215.714,Z 754.64,A -85,B 0,C 180,E1 5743.853,E2 5743.853} C_VEL
LIN {X 0,Y 202.493,Z 769.073,A -85,B 0,C 180,E1 5741.445,E2 5741.445} C_VEL
LIN {X 0,Y 187.417,Z 783.845,A -85,B 0,C 180,E1 5738.164,E2 5738.164} C_VEL
LIN {X 0,Y 173.066,Z 796.312,A -85,B 0,C 180,E1 5734.321,E2 5734.321} C_VEL
LIN {X 0,Y 159.638,Z 807.035,A -85,B 0,C 180,E1 5729.804,E2 5729.804} C_VEL
LIN {X 0,Y 145.424,Z 817.416,A -85,B 0,C 180,E1 5723.553,E2 5723.553} C_VEL
LIN {X 0,Y 134.813,Z 824.746,A -85,B 0,C 180,E1 5717.242,E2 5717.242} C_VEL
LIN {X 0,Y 124.697,Z 831.701,A -85,B 0,C 180,E1 5708.712,E2 5708.712} C_VEL
LIN {X 0,Y 117.117,Z 837.041,A -85,B 0,C 180,E1 5698.438,E2 5698.438} C_VEL
LIN {X 0,Y 113.433,Z 840.203,A -85,B 0,C 180,E1 5689.034,E2 5689.034} C_VEL
LIN {X 0,Y 112.215,Z 841.758,A -85,B 0,C 180,E1 5681.623,E2 5681.623} C_VEL
LIN {X 0,Y 111.118,Z 842.322,A -85,B 0,C 180,E1 5677.979,E2 5677.979} C_VEL
LIN {X 0,Y 108.09,Z 842.534,A -85,B 0,C 180,E1 5672.959,E2 5672.959} C_VEL
LIN {X 0,Y 104.182,Z 842.31,A -85,B 0,C 180,E1 5664.912,E2 5664.912} C_VEL
LIN {X 0,Y 104.02,Z 842.193,A -85,B 0,C 180,E1 5663.035,E2 5663.035} C_VEL
LIN {X 0,Y 105.19,Z 840.516,A -85,B 0,C 180,E1 5651.72,E2 5651.72} C_VEL
LIN {X 0,Y 109.154,Z 837.337,A -85,B 0,C 180,E1 5640.957,E2 5640.957} C_VEL
LIN {X 0,Y 116.154,Z 832.77,A -85,B 0,C 180,E1 5631.07,E2 5631.07} C_VEL
LIN {X 0,Y 127.779,Z 825.49,A -85,B 0,C 180,E1 5621.094,E2 5621.094} C_VEL
LIN {X 0,Y 139.319,Z 818.029,A -85,B 0,C 180,E1 5614.381,E2 5614.381} C_VEL
LIN {X 0,Y 153.398,Z 808.441,A -85,B 0,C 180,E1 5608.368,E2 5608.368} C_VEL
LIN {X 0,Y 168.044,Z 797.339,A -85,B 0,C 180,E1 5603.613,E2 5603.613} C_VEL
LIN {X 0,Y 182.972,Z 784.924,A -85,B 0,C 180,E1 5599.804,E2 5599.804} C_VEL
LIN {X 0,Y 199.151,Z 769.714,A -85,B 0,C 180,E1 5596.483,E2 5596.483} C_VEL
LIN {X 0,Y 212.951,Z 755.083,A -85,B 0,C 180,E1 5594.132,E2 5594.132} C_VEL
LIN {X 0,Y 227.534,Z 737.504,A -85,B 0,C 180,E1 5592.029,E2 5592.029} C_VEL
LIN {X 0,Y 239.492,Z 720.893,A -85,B 0,C 180,E1 5590.529,E2 5590.529} C_VEL
LIN {X 0,Y 251.215,Z 702.278,A -85,B 0,C 180,E1 5589.236,E2 5589.236} C_VEL
LIN {X 0,Y 261.63,Z 682.648,A -85,B 0,C 180,E1 5588.199,E2 5588.199} C_VEL
LIN {X 0,Y 269.995,Z 664.094,A -85,B 0,C 180,E1 5587.447,E2 5587.447} C_VEL
LIN {X 0,Y 278.146,Z 641.944,A -85,B 0,C 180,E1 5586.777,E2 5586.777} C_VEL
LIN {X 0,Y 284.382,Z 619.783,A -85,B 0,C 180,E1 5586.29,E2 5586.29} C_VEL
LIN {X 0,Y 289.192,Z 595.532,A -85,B 0,C 180,E1 5585.85,E2 5585.85} C_VEL
LIN {X 0,Y 298.119,Z 520.506,A -85,B 0,C 180,E1 5584.66,E2 5584.66} C_VEL
LIN {X 0,Y 297.79,Z 519.399,A -85,B 0,C 180,E1 5583.465,E2 5583.465} C_VEL
LIN {X 0,Y 297.311,Z 518.337,A -85,B 0,C 180,E1 5579.422,E2 5579.422} C_VEL
LIN {X 0,Y 297.96,Z 519.845,A -85,B 0,C 180,E1 5575.477,E2 5575.477} C_VEL
LIN {X 0,Y 299.099,Z 523.324,A -85,B 0,C 180,E1 5572.509,E2 5572.509} C_VEL
LIN {X 0,Y 305.801,Z 534.476,A -85,B 0,C 180,E1 5564.74,E2 5564.74} C_VEL
LIN {X 0,Y 310.788,Z 538.638,A -85,B 0,C 180,E1 5561.331,E2 5561.331} C_VEL
LIN {X 0,Y 316.37,Z 543.05,A -85,B 0,C 180,E1 5557.908,E2 5557.908} C_VEL
LIN {X 0,Y 321.107,Z 545.974,A -85,B 0,C 180,E1 5554.749,E2 5554.749} C_VEL
LIN {X 0,Y 323.098,Z 547.5,A -85,B 0,C 180,E1 5553.239,E2 5553.239} C_VEL
LIN {X 0,Y 326.841,Z 550.954,A -85,B 0,C 180,E1 5550.09,E2 5550.09} C_VEL
LIN {X 0,Y 330.321,Z 553.649,A -85,B 0,C 180,E1 5546.658,E2 5546.658} C_VEL
LIN {X 0,Y 331.68,Z 554.858,A -85,B 0,C 180,E1 5545.268,E2 5545.268} C_VEL
LIN {X 0,Y 334.875,Z 558.429,A -85,B 0,C 180,E1 5541.742,E2 5541.742} C_VEL
LIN {X 0,Y 338.254,Z 560.987,A -85,B 0,C 180,E1 5538.084,E2 5538.084} C_VEL
LIN {X 0,Y 339.652,Z 562.11,A -85,B 0,C 180,E1 5536.462,E2 5536.462} C_VEL
LIN {X 0,Y 342.624,Z 565.534,A -85,B 0,C 180,E1 5532.838,E2 5532.838} C_VEL
LIN {X 0,Y 345.39,Z 567.797,A -85,B 0,C 180,E1 5529.343,E2 5529.343} C_VEL
LIN {X 0,Y 348.139,Z 569.533,A -85,B 0,C 180,E1 5525.755,E2 5525.755} C_VEL
LIN {X 0,Y 350.505,Z 572.63,A -85,B 0,C 180,E1 5522.089,E2 5522.089} C_VEL
LIN {X 0,Y 352.769,Z 574.669,A -85,B 0,C 180,E1 5518.434,E2 5518.434} C_VEL
LIN {X 0,Y 354.923,Z 575.982,A -85,B 0,C 180,E1 5514.64,E2 5514.64} C_VEL
LIN {X 0,Y 356.862,Z 576.876,A -85,B 0,C 180,E1 5510.844,E2 5510.844} C_VEL
LIN {X 0,Y 358.134,Z 578.857,A -85,B 0,C 180,E1 5507.381,E2 5507.381} C_VEL
LIN {X 0,Y 359.344,Z 580.433,A -85,B 0,C 180,E1 5503.68,E2 5503.68} C_VEL
LIN {X 0,Y 360.162,Z 581.337,A -85,B 0,C 180,E1 5500.396,E2 5500.396} C_VEL
LIN {X 0,Y 360.885,Z 581.94,A -85,B 0,C 180,E1 5496.682,E2 5496.682} C_VEL
LIN {X 0,Y 361.226,Z 582.21,A -85,B 0,C 180,E1 5493.332,E2 5493.332} C_VEL
LIN {X 0,Y 361.389,Z 582.32,A -85,B 0,C 180,E1 5489.683,E2 5489.683} C_VEL
LIN {X 0,Y 361.196,Z 582.209,A -85,B 0,C 180,E1 5486.35,E2 5486.35} C_VEL
LIN {X 0,Y 360.832,Z 581.848,A -85,B 0,C 180,E1 5482.752,E2 5482.752} C_VEL
LIN {X 0,Y 360.083,Z 581.263,A -85,B 0,C 180,E1 5479.278,E2 5479.278} C_VEL
LIN {X 0,Y 359.17,Z 580.187,A -85,B 0,C 180,E1 5475.641,E2 5475.641} C_VEL
LIN {X 0,Y 357.999,Z 578.676,A -85,B 0,C 180,E1 5472.247,E2 5472.247} C_VEL
LIN {X 0,Y 356.711,Z 576.749,A -85,B 0,C 180,E1 5468.803,E2 5468.803} C_VEL
LIN {X 0,Y 354.809,Z 575.922,A -85,B 0,C 180,E1 5465.148,E2 5465.148} C_VEL
LIN {X 0,Y 352.653,Z 574.586,A -85,B 0,C 180,E1 5461.371,E2 5461.371} C_VEL
LIN {X 0,Y 350.27,Z 572.374,A -85,B 0,C 180,E1 5457.545,E2 5457.545} C_VEL
LIN {X 0,Y 347.674,Z 569.062,A -85,B 0,C 180,E1 5453.633,E2 5453.633} C_VEL
LIN {X 0,Y 345.026,Z 567.538,A -85,B 0,C 180,E1 5450.17,E2 5450.17} C_VEL
LIN {X 0,Y 342.035,Z 564.954,A -85,B 0,C 180,E1 5446.466,E2 5446.466} C_VEL
LIN {X 0,Y 338.962,Z 561.391,A -85,B 0,C 180,E1 5442.722,E2 5442.722} C_VEL
LIN {X 0,Y 335.527,Z 558.985,A -85,B 0,C 180,E1 5438.945,E2 5438.945} C_VEL
LIN {X 0,Y 332.349,Z 555.76,A -85,B 0,C 180,E1 5435.495,E2 5435.495} C_VEL
LIN {X 0,Y 330.759,Z 553.908,A -85,B 0,C 180,E1 5433.77,E2 5433.77} C_VEL
LIN {X 0,Y 327.394,Z 551.444,A -85,B 0,C 180,E1 5430.462,E2 5430.462} C_VEL
LIN {X 0,Y 323.669,Z 548.068,A -85,B 0,C 180,E1 5427.206,E2 5427.206} C_VEL
LIN {X 0,Y 321.588,Z 546.228,A -85,B 0,C 180,E1 5425.605,E2 5425.605} C_VEL
LIN {X 0,Y 316.907,Z 543.432,A -85,B 0,C 180,E1 5422.443,E2 5422.443} C_VEL
LIN {X 0,Y 311.661,Z 539.409,A -85,B 0,C 180,E1 5419.198,E2 5419.198} C_VEL
LIN {X 0,Y 307.906,Z 536.264,A -85,B 0,C 180,E1 5416.799,E2 5416.799} C_VEL
LIN {X 0,Y 302.802,Z 530.809,A -85,B 0,C 180,E1 5412.588,E2 5412.588} C_VEL
LIN {X 0,Y 300.129,Z 525.963,A -85,B 0,C 180,E1 5409.298,E2 5409.298} C_VEL
LIN {X 0,Y 298.58,Z 521.838,A -85,B 0,C 180,E1 5406.345,E2 5406.345} C_VEL
LIN {X 0,Y 297.775,Z 519.376,A -85,B 0,C 180,E1 5403.851,E2 5403.851} C_VEL
LIN {X 0,Y 297.308,Z 518.329,A -85,B 0,C 180,E1 5400,E2 5400} C_VEL
LIN {X 0,Y 297.949,Z 519.793,A -85,B 0,C 180,E1 5395.959,E2 5395.959} C_VEL
LIN {X 0,Y 298.107,Z 520.666,A -85,B 0,C 180,E1 5395.321,E2 5395.321} C_VEL
LIN {X 0,Y 289.028,Z 596.616,A -85,B 0,C 180,E1 5394.132,E2 5394.132} C_VEL
LIN {X 0,Y 284.232,Z 620.381,A -85,B 0,C 180,E1 5393.699,E2 5393.699} C_VEL
LIN {X 0,Y 277.905,Z 642.699,A -85,B 0,C 180,E1 5393.205,E2 5393.205} C_VEL
LIN {X 0,Y 269.743,Z 664.688,A -85,B 0,C 180,E1 5392.532,E2 5392.532} C_VEL
LIN {X 0,Y 261.63,Z 682.647,A -85,B 0,C 180,E1 5391.801,E2 5391.801} C_VEL
LIN {X 0,Y 250.794,Z 703.005,A -85,B 0,C 180,E1 5390.719,E2 5390.719} C_VEL
LIN {X 0,Y 239.027,Z 721.58,A -85,B 0,C 180,E1 5389.416,E2 5389.416} C_VEL
LIN {X 0,Y 226.09,Z 739.412,A -85,B 0,C 180,E1 5387.774,E2 5387.774} C_VEL
LIN {X 0,Y 212.015,Z 756.118,A -85,B 0,C 180,E1 5385.721,E2 5385.721} C_VEL
LIN {X 0,Y 198.277,Z 770.605,A -85,B 0,C 180,E1 5383.354,E2 5383.354} C_VEL
LIN {X 0,Y 181.978,Z 785.771,A -85,B 0,C 180,E1 5379.97,E2 5379.97} C_VEL
LIN {X 0,Y 167.247,Z 797.98,A -85,B 0,C 180,E1 5376.157,E2 5376.157} C_VEL
LIN {X 0,Y 151.187,Z 809.947,A -85,B 0,C 180,E1 5370.803,E2 5370.803} C_VEL
LIN {X 0,Y 138.587,Z 818.51,A -85,B 0,C 180,E1 5365.253,E2 5365.253} C_VEL
LIN {X 0,Y 125.777,Z 826.807,A -85,B 0,C 180,E1 5357.491,E2 5357.491} C_VEL
LIN {X 0,Y 115.323,Z 833.278,A -85,B 0,C 180,E1 5347.992,E2 5347.992} C_VEL
LIN {X 0,Y 108.62,Z 837.732,A -85,B 0,C 180,E1 5337.998,E2 5337.998} C_VEL
LIN {X 0,Y 104.664,Z 841.044,A -85,B 0,C 180,E1 5325.514,E2 5325.514} C_VEL
LIN {X 0,Y 104.013,Z 842.242,A -85,B 0,C 180,E1 5316.07,E2 5316.07} C_VEL
LIN {X 0,Y 104.046,Z 842.502,A -85,B 0,C 180,E1 5308.899,E2 5308.899} C_VEL
LIN {X 0,Y 104.02,Z 842.193,A -85,B 0,C 180,E1 5303.035,E2 5303.035} C_VEL
LIN {X 0,Y 103.331,Z 841.82,A -85,B 0,C 180,E1 5299.084,E2 5299.084} C_VEL
LIN {X 0,Y 100.655,Z 840.739,A -85,B 0,C 180,E1 5292.682,E2 5292.682} C_VEL
LIN {X 0,Y 99.185,Z 839.242,A -85,B 0,C 180,E1 5285.991,E2 5285.991} C_VEL
LIN {X 0,Y 99.841,Z 838.548,A -85,B 0,C 180,E1 5283.135,E2 5283.135} C_VEL
LIN {X 0,Y 107.182,Z 834.041,A -85,B 0,C 180,E1 5271.318,E2 5271.318} C_VEL
LIN {X 0,Y 117.025,Z 828.391,A -85,B 0,C 180,E1 5261.986,E2 5261.986} C_VEL
LIN {X 0,Y 130.931,Z 820.214,A -85,B 0,C 180,E1 5253.355,E2 5253.355} C_VEL
LIN {X 0,Y 144.279,Z 811.689,A -85,B 0,C 180,E1 5247.499,E2 5247.499} C_VEL
LIN {X 0,Y 159.167,Z 801.415,A -85,B 0,C 180,E1 5242.572,E2 5242.572} C_VEL
LIN {X 0,Y 175.873,Z 788.391,A -85,B 0,C 180,E1 5238.307,E2 5238.307} C_VEL
LIN {X 0,Y 190.722,Z 775.418,A -85,B 0,C 180,E1 5235.293,E2 5235.293} C_VEL
LIN {X 0,Y 207.298,Z 758.958,A -85,B 0,C 180,E1 5232.536,E2 5232.536} C_VEL
LIN {X 0,Y 221.703,Z 742.569,A -85,B 0,C 180,E1 5230.54,E2 5230.54} C_VEL
LIN {X 0,Y 236.248,Z 723.393,A -85,B 0,C 180,E1 5228.811,E2 5228.811} C_VEL
LIN {X 0,Y 247.604,Z 706.054,A -85,B 0,C 180,E1 5227.637,E2 5227.637} C_VEL
LIN {X 0,Y 258.676,Z 686.344,A -85,B 0,C 180,E1 5226.611,E2 5226.611} C_VEL
LIN {X 0,Y 267.845,Z 666.708,A -85,B 0,C 180,E1 5225.84,E2 5225.84} C_VEL
LIN {X 0,Y 275.851,Z 646.019,A -85,B 0,C 180,E1 5225.229,E2 5225.229} C_VEL
LIN {X 0,Y 282.568,Z 623.649,A -85,B 0,C 180,E1 5224.751,E2 5224.751} C_VEL
LIN {X 0,Y 287.417,Z 601.724,A -85,B 0,C 180,E1 5224.367,E2 5224.367} C_VEL
LIN {X 0,Y 291.679,Z 570.225,A -85,B 0,C 180,E1 5223.879,E2 5223.879} C_VEL
LIN {X 0,Y 296.741,Z 527.263,A -85,B 0,C 180,E1 5223.214,E2 5223.214} C_VEL
LIN {X 0,Y 296.336,Z 526.279,A -85,B 0,C 180,E1 5219.42,E2 5219.42} C_VEL
LIN {X 0,Y 296.917,Z 527.762,A -85,B 0,C 180,E1 5215.655,E2 5215.655} C_VEL
LIN {X 0,Y 297.957,Z 531.166,A -85,B 0,C 180,E1 5212.771,E2 5212.771} C_VEL
LIN {X 0,Y 304.376,Z 542.168,A -85,B 0,C 180,E1 5205.056,E2 5205.056} C_VEL
LIN {X 0,Y 309.406,Z 546.458,A -85,B 0,C 180,E1 5201.537,E2 5201.537} C_VEL
LIN {X 0,Y 315.159,Z 550.96,A -85,B 0,C 180,E1 5198.015,E2 5198.015} C_VEL
LIN {X 0,Y 319.923,Z 553.869,A -85,B 0,C 180,E1 5194.847,E2 5194.847} C_VEL
LIN {X 0,Y 321.93,Z 555.458,A -85,B 0,C 180,E1 5193.334,E2 5193.334} C_VEL
LIN {X 0,Y 325.512,Z 558.708,A -85,B 0,C 180,E1 5190.361,E2 5190.361} C_VEL
LIN {X 0,Y 329.14,Z 561.496,A -85,B 0,C 180,E1 5186.852,E2 5186.852} C_VEL
LIN {X 0,Y 330.603,Z 562.839,A -85,B 0,C 180,E1 5185.346,E2 5185.346} C_VEL
LIN {X 0,Y 333.924,Z 566.46,A -85,B 0,C 180,E1 5181.698,E2 5181.698} C_VEL
LIN {X 0,Y 337.378,Z 569.014,A -85,B 0,C 180,E1 5177.95,E2 5177.95} C_VEL
LIN {X 0,Y 338.688,Z 570.202,A -85,B 0,C 180,E1 5176.423,E2 5176.423} C_VEL
LIN {X 0,Y 341.705,Z 573.605,A -85,B 0,C 180,E1 5172.74,E2 5172.74} C_VEL
LIN {X 0,Y 344.515,Z 575.827,A -85,B 0,C 180,E1 5169.205,E2 5169.205} C_VEL
LIN {X 0,Y 347.123,Z 577.527,A -85,B 0,C 180,E1 5165.782,E2 5165.782} C_VEL
LIN {X 0,Y 349.496,Z 580.577,A -85,B 0,C 180,E1 5162.133,E2 5162.133} C_VEL
LIN {X 0,Y 351.729,Z 582.582,A -85,B 0,C 180,E1 5158.526,E2 5158.526} C_VEL
LIN {X 0,Y 353.905,Z 583.906,A -85,B 0,C 180,E1 5154.716,E2 5154.716} C_VEL
LIN {X 0,Y 355.865,Z 584.804,A -85,B 0,C 180,E1 5150.905,E2 5150.905} C_VEL
LIN {X 0,Y 357.172,Z 586.837,A -85,B 0,C 180,E1 5147.334,E2 5147.334} C_VEL
LIN {X 0,Y 358.359,Z 588.371,A -85,B 0,C 180,E1 5143.719,E2 5143.719} C_VEL
LIN {X 0,Y 359.221,Z 589.307,A -85,B 0,C 180,E1 5140.261,E2 5140.261} C_VEL
LIN {X 0,Y 359.928,Z 589.927,A -85,B 0,C 180,E1 5136.38,E2 5136.38} C_VEL
LIN {X 0,Y 360.269,Z 590.153,A -85,B 0,C 180,E1 5133.182,E2 5133.182} C_VEL
LIN {X 0,Y 360.383,Z 590.243,A -85,B 0,C 180,E1 5129.364,E2 5129.364} C_VEL
LIN {X 0,Y 360.209,Z 590.146,A -85,B 0,C 180,E1 5126.18,E2 5126.18} C_VEL
LIN {X 0,Y 359.787,Z 589.751,A -85,B 0,C 180,E1 5122.495,E2 5122.495} C_VEL
LIN {X 0,Y 359.065,Z 589.16,A -85,B 0,C 180,E1 5119.085,E2 5119.085} C_VEL
LIN {X 0,Y 358.045,Z 588.016,A -85,B 0,C 180,E1 5115.279,E2 5115.279} C_VEL
LIN {X 0,Y 356.956,Z 586.54,A -85,B 0,C 180,E1 5112.055,E2 5112.055} C_VEL
LIN {X 0,Y 355.693,Z 584.677,A -85,B 0,C 180,E1 5108.739,E2 5108.739} C_VEL
LIN {X 0,Y 353.806,Z 583.853,A -85,B 0,C 180,E1 5105.098,E2 5105.098} C_VEL
LIN {X 0,Y 351.615,Z 582.499,A -85,B 0,C 180,E1 5101.278,E2 5101.278} C_VEL
LIN {X 0,Y 349.32,Z 580.397,A -85,B 0,C 180,E1 5097.605,E2 5097.605} C_VEL
LIN {X 0,Y 346.794,Z 577.085,A -85,B 0,C 180,E1 5093.77,E2 5093.77} C_VEL
LIN {X 0,Y 343.912,Z 575.416,A -85,B 0,C 180,E1 5090.022,E2 5090.022} C_VEL
LIN {X 0,Y 340.991,Z 572.901,A -85,B 0,C 180,E1 5086.407,E2 5086.407} C_VEL
LIN {X 0,Y 337.789,Z 569.248,A -85,B 0,C 180,E1 5082.522,E2 5082.522} C_VEL
LIN {X 0,Y 334.276,Z 566.763,A -85,B 0,C 180,E1 5078.679,E2 5078.679} C_VEL
LIN {X 0,Y 330.942,Z 563.291,A -85,B 0,C 180,E1 5075.032,E2 5075.032} C_VEL
LIN {X 0,Y 329.408,Z 561.662,A -85,B 0,C 180,E1 5073.416,E2 5073.416} C_VEL
LIN {X 0,Y 325.933,Z 559.042,A -85,B 0,C 180,E1 5070.002,E2 5070.002} C_VEL
LIN {X 0,Y 322.155,Z 555.683,A -85,B 0,C 180,E1 5066.845,E2 5066.845} C_VEL
LIN {X 0,Y 320.188,Z 554,A -85,B 0,C 180,E1 5065.329,E2 5065.329} C_VEL
LIN {X 0,Y 315.427,Z 551.151,A -85,B 0,C 180,E1 5062.161,E2 5062.161} C_VEL
LIN {X 0,Y 309.69,Z 546.72,A -85,B 0,C 180,E1 5058.64,E2 5058.64} C_VEL
LIN {X 0,Y 306.053,Z 543.668,A -85,B 0,C 180,E1 5056.22,E2 5056.22} C_VEL
LIN {X 0,Y 301.199,Z 538.074,A -85,B 0,C 180,E1 5051.974,E2 5051.974} C_VEL
LIN {X 0,Y 297.593,Z 529.928,A -85,B 0,C 180,E1 5046.366,E2 5046.366} C_VEL
LIN {X 0,Y 296.747,Z 527.265,A -85,B 0,C 180,E1 5043.67,E2 5043.67} C_VEL
LIN {X 0,Y 296.337,Z 526.279,A -85,B 0,C 180,E1 5039.807,E2 5039.807} C_VEL
LIN {X 0,Y 296.721,Z 527.497,A -85,B 0,C 180,E1 5036.758,E2 5036.758} C_VEL
LIN {X 0,Y 288.287,Z 596.566,A -85,B 0,C 180,E1 5035.717,E2 5035.717} C_VEL
LIN {X 0,Y 283.432,Z 620.261,A -85,B 0,C 180,E1 5035.311,E2 5035.311} C_VEL
LIN {X 0,Y 277.069,Z 642.442,A -85,B 0,C 180,E1 5034.856,E2 5034.856} C_VEL
LIN {X 0,Y 269.298,Z 663.313,A -85,B 0,C 180,E1 5034.274,E2 5034.274} C_VEL
LIN {X 0,Y 261.081,Z 681.412,A -85,B 0,C 180,E1 5033.605,E2 5033.605} C_VEL
LIN {X 0,Y 250.567,Z 701.13,A -85,B 0,C 180,E1 5032.65,E2 5032.65} C_VEL
LIN {X 0,Y 238.613,Z 719.957,A -85,B 0,C 180,E1 5031.448,E2 5031.448} C_VEL
LIN {X 0,Y 226.369,Z 736.732,A -85,B 0,C 180,E1 5030.047,E2 5030.047} C_VEL
LIN {X 0,Y 211.521,Z 754.377,A -85,B 0,C 180,E1 5028.087,E2 5028.087} C_VEL
LIN {X 0,Y 197.86,Z 768.582,A -85,B 0,C 180,E1 5025.962,E2 5025.962} C_VEL
LIN {X 0,Y 181.928,Z 783.329,A -85,B 0,C 180,E1 5022.991,E2 5022.991} C_VEL
LIN {X 0,Y 166.569,Z 795.805,A -85,B 0,C 180,E1 5019.454,E2 5019.454} C_VEL
LIN {X 0,Y 151.976,Z 806.524,A -85,B 0,C 180,E1 5015.214,E2 5015.214} C_VEL
LIN {X 0,Y 135.764,Z 817.186,A -85,B 0,C 180,E1 5008.967,E2 5008.967} C_VEL
LIN {X 0,Y 122.908,Z 824.98,A -85,B 0,C 180,E1 5002.099,E2 5002.099} C_VEL
LIN {X 0,Y 110.31,Z 832.261,A -85,B 0,C 180,E1 4992.123,E2 4992.123} C_VEL
LIN {X 0,Y 102.308,Z 836.914,A -85,B 0,C 180,E1 4981.761,E2 4981.761} C_VEL
LIN {X 0,Y 97.622,Z 840.124,A -85,B 0,C 180,E1 4970.379,E2 4970.379} C_VEL
LIN {X 0,Y 96.049,Z 841.902,A -85,B 0,C 180,E1 4958.38,E2 4958.38} C_VEL
LIN {X 0,Y 96.066,Z 842.297,A -85,B 0,C 180,E1 4950,E2 4950} C_VEL
LIN {X 0,Y 96.064,Z 841.87,A -85,B 0,C 180,E1 4941.018,E2 4941.018} C_VEL
LIN {X 0,Y 97.947,Z 839.841,A -85,B 0,C 180,E1 4928.44,E2 4928.44} C_VEL
LIN {X 0,Y 99.841,Z 838.548,A -85,B 0,C 180,E1 4923.135,E2 4923.135} C_VEL
LIN {X 0,Y 100.931,Z 837.369,A -85,B 0,C 180,E1 4918.796,E2 4918.796} C_VEL
LIN {X 0,Y 102.848,Z 833.151,A -85,B 0,C 180,E1 4907.089,E2 4907.089} C_VEL
LIN {X 0,Y 105.411,Z 831.469,A -85,B 0,C 180,E1 4903.823,E2 4903.823} C_VEL
LIN {X 0,Y 118.657,Z 824.353,A -85,B 0,C 180,E1 4894.334,E2 4894.334} C_VEL
LIN {X 0,Y 132.166,Z 816.649,A -85,B 0,C 180,E1 4887.736,E2 4887.736} C_VEL
LIN {X 0,Y 149.92,Z 805.423,A -85,B 0,C 180,E1 4881.519,E2 4881.519} C_VEL
LIN {X 0,Y 165.581,Z 794.271,A -85,B 0,C 180,E1 4877.436,E2 4877.436} C_VEL
LIN {X 0,Y 182.696,Z 780.499,A -85,B 0,C 180,E1 4873.934,E2 4873.934} C_VEL
LIN {X 0,Y 196.964,Z 767.42,A -85,B 0,C 180,E1 4871.562,E2 4871.562} C_VEL
LIN {X 0,Y 212.329,Z 751.584,A -85,B 0,C 180,E1 4869.423,E2 4869.423} C_VEL
LIN {X 0,Y 227.006,Z 734.019,A -85,B 0,C 180,E1 4867.696,E2 4867.696} C_VEL
LIN {X 0,Y 239.464,Z 716.959,A -85,B 0,C 180,E1 4866.427,E2 4866.427} C_VEL
LIN {X 0,Y 252.034,Z 696.738,A -85,B 0,C 180,E1 4865.299,E2 4865.299} C_VEL
LIN {X 0,Y 261.767,Z 678.202,A -85,B 0,C 180,E1 4864.513,E2 4864.513} C_VEL
LIN {X 0,Y 271.062,Z 657.022,A -85,B 0,C 180,E1 4863.839,E2 4863.839} C_VEL
LIN {X 0,Y 278.43,Z 635.989,A -85,B 0,C 180,E1 4863.353,E2 4863.353} C_VEL
LIN {X 0,Y 284.575,Z 613.084,A -85,B 0,C 180,E1 4862.952,E2 4862.952} C_VEL
LIN {X 0,Y 288.508,Z 591.284,A -85,B 0,C 180,E1 4862.613,E2 4862.613} C_VEL
LIN {X 0,Y 295.481,Z 534.677,A -85,B 0,C 180,E1 4861.793,E2 4861.793} C_VEL
LIN {X 0,Y 295.372,Z 534.288,A -85,B 0,C 180,E1 4859.03,E2 4859.03} C_VEL
LIN {X 0,Y 295.878,Z 535.678,A -85,B 0,C 180,E1 4855.834,E2 4855.834} C_VEL
LIN {X 0,Y 296.782,Z 538.86,A -85,B 0,C 180,E1 4853.131,E2 4853.131} C_VEL
LIN {X 0,Y 302.959,Z 549.86,A -85,B 0,C 180,E1 4845.376,E2 4845.376} C_VEL
LIN {X 0,Y 308.028,Z 554.279,A -85,B 0,C 180,E1 4841.746,E2 4841.746} C_VEL
LIN {X 0,Y 313.948,Z 558.869,A -85,B 0,C 180,E1 4838.123,E2 4838.123} C_VEL
LIN {X 0,Y 318.469,Z 561.63,A -85,B 0,C 180,E1 4835.121,E2 4835.121} C_VEL
LIN {X 0,Y 320.545,Z 563.184,A -85,B 0,C 180,E1 4833.609,E2 4833.609} C_VEL
LIN {X 0,Y 324.157,Z 566.458,A -85,B 0,C 180,E1 4830.631,E2 4830.631} C_VEL
LIN {X 0,Y 327.884,Z 569.291,A -85,B 0,C 180,E1 4827.126,E2 4827.126} C_VEL
LIN {X 0,Y 329.429,Z 570.695,A -85,B 0,C 180,E1 4825.525,E2 4825.525} C_VEL
LIN {X 0,Y 332.707,Z 574.257,A -85,B 0,C 180,E1 4821.938,E2 4821.938} C_VEL
LIN {X 0,Y 336.14,Z 576.83,A -85,B 0,C 180,E1 4818.218,E2 4818.218} C_VEL
LIN {X 0,Y 337.552,Z 578.065,A -85,B 0,C 180,E1 4816.591,E2 4816.591} C_VEL
LIN {X 0,Y 340.577,Z 581.448,A -85,B 0,C 180,E1 4812.928,E2 4812.928} C_VEL
LIN {X 0,Y 343.567,Z 583.807,A -85,B 0,C 180,E1 4809.161,E2 4809.161} C_VEL
LIN {X 0,Y 346.03,Z 585.42,A -85,B 0,C 180,E1 4805.913,E2 4805.913} C_VEL
LIN {X 0,Y 348.423,Z 588.467,A -85,B 0,C 180,E1 4802.259,E2 4802.259} C_VEL
LIN {X 0,Y 350.709,Z 590.508,A -85,B 0,C 180,E1 4798.587,E2 4798.587} C_VEL
LIN {X 0,Y 352.887,Z 591.829,A -85,B 0,C 180,E1 4794.792,E2 4794.792} C_VEL
LIN {X 0,Y 354.867,Z 592.732,A -85,B 0,C 180,E1 4790.966,E2 4790.966} C_VEL
LIN {X 0,Y 356.182,Z 594.782,A -85,B 0,C 180,E1 4787.363,E2 4787.363} C_VEL
LIN {X 0,Y 357.374,Z 596.309,A -85,B 0,C 180,E1 4783.757,E2 4783.757} C_VEL
LIN {X 0,Y 358.238,Z 597.244,A -85,B 0,C 180,E1 4780.289,E2 4780.289} C_VEL
LIN {X 0,Y 358.951,Z 597.866,A -85,B 0,C 180,E1 4776.397,E2 4776.397} C_VEL
LIN {X 0,Y 359.293,Z 598.093,A -85,B 0,C 180,E1 4773.19,E2 4773.19} C_VEL
LIN {X 0,Y 359.408,Z 598.184,A -85,B 0,C 180,E1 4769.362,E2 4769.362} C_VEL
LIN {X 0,Y 359.234,Z 598.086,A -85,B 0,C 180,E1 4766.17,E2 4766.17} C_VEL
LIN {X 0,Y 358.806,Z 597.69,A -85,B 0,C 180,E1 4762.474,E2 4762.474} C_VEL
LIN {X 0,Y 358.082,Z 597.098,A -85,B 0,C 180,E1 4759.055,E2 4759.055} C_VEL
LIN {X 0,Y 357.052,Z 595.95,A -85,B 0,C 180,E1 4755.237,E2 4755.237} C_VEL
LIN {X 0,Y 355.961,Z 594.476,A -85,B 0,C 180,E1 4752.003,E2 4752.003} C_VEL
LIN {X 0,Y 354.676,Z 592.606,A -85,B 0,C 180,E1 4748.675,E2 4748.675} C_VEL
LIN {X 0,Y 352.79,Z 591.777,A -85,B 0,C 180,E1 4745.022,E2 4745.022} C_VEL
LIN {X 0,Y 350.579,Z 590.412,A -85,B 0,C 180,E1 4741.185,E2 4741.185} C_VEL
LIN {X 0,Y 348.284,Z 588.325,A -85,B 0,C 180,E1 4737.532,E2 4737.532} C_VEL
LIN {X 0,Y 345.803,Z 585.115,A -85,B 0,C 180,E1 4733.775,E2 4733.775} C_VEL
LIN {X 0,Y 342.956,Z 583.398,A -85,B 0,C 180,E1 4730.063,E2 4730.063} C_VEL
LIN {X 0,Y 339.947,Z 580.847,A -85,B 0,C 180,E1 4726.347,E2 4726.347} C_VEL
LIN {X 0,Y 336.679,Z 577.137,A -85,B 0,C 180,E1 4722.387,E2 4722.387} C_VEL
LIN {X 0,Y 333.226,Z 574.703,A -85,B 0,C 180,E1 4718.617,E2 4718.617} C_VEL
LIN {X 0,Y 329.862,Z 571.258,A -85,B 0,C 180,E1 4714.952,E2 4714.952} C_VEL
LIN {X 0,Y 328.251,Z 569.526,A -85,B 0,C 180,E1 4713.249,E2 4713.249} C_VEL
LIN {X 0,Y 324.601,Z 566.797,A -85,B 0,C 180,E1 4709.731,E2 4709.731} C_VEL
LIN {X 0,Y 320.876,Z 563.523,A -85,B 0,C 180,E1 4706.661,E2 4706.661} C_VEL
LIN {X 0,Y 318.731,Z 561.763,A -85,B 0,C 180,E1 4705.055,E2 4705.055} C_VEL
LIN {X 0,Y 314.216,Z 559.058,A -85,B 0,C 180,E1 4702.054,E2 4702.054} C_VEL
LIN {X 0,Y 308.168,Z 554.409,A -85,B 0,C 180,E1 4698.344,E2 4698.344} C_VEL
LIN {X 0,Y 304.232,Z 551.059,A -85,B 0,C 180,E1 4695.634,E2 4695.634} C_VEL
LIN {X 0,Y 299.554,Z 545.185,A -85,B 0,C 180,E1 4691.26,E2 4691.26} C_VEL
LIN {X 0,Y 296.297,Z 537.243,A -85,B 0,C 180,E1 4685.616,E2 4685.616} C_VEL
LIN {X 0,Y 295.722,Z 535.153,A -85,B 0,C 180,E1 4683.489,E2 4683.489} C_VEL
LIN {X 0,Y 295.362,Z 534.224,A -85,B 0,C 180,E1 4679.806,E2 4679.806} C_VEL
LIN {X 0,Y 295.462,Z 534.836,A -85,B 0,C 180,E1 4678.201,E2 4678.201} C_VEL
LIN {X 0,Y 287.738,Z 596.71,A -85,B 0,C 180,E1 4677.306,E2 4677.306} C_VEL
LIN {X 0,Y 282.827,Z 620.261,A -85,B 0,C 180,E1 4676.928,E2 4676.928} C_VEL
LIN {X 0,Y 276.218,Z 642.902,A -85,B 0,C 180,E1 4676.501,E2 4676.501} C_VEL
LIN {X 0,Y 268.075,Z 664.313,A -85,B 0,C 180,E1 4675.948,E2 4675.948} C_VEL
LIN {X 0,Y 259.33,Z 683.137,A -85,B 0,C 180,E1 4675.295,E2 4675.295} C_VEL
LIN {X 0,Y 247.907,Z 703.811,A -85,B 0,C 180,E1 4674.342,E2 4674.342} C_VEL
LIN {X 0,Y 236.098,Z 721.769,A -85,B 0,C 180,E1 4673.247,E2 4673.247} C_VEL
LIN {X 0,Y 222.252,Z 740.042,A -85,B 0,C 180,E1 4671.769,E2 4671.769} C_VEL
LIN {X 0,Y 208.109,Z 756.114,A -85,B 0,C 180,E1 4670.028,E2 4670.028} C_VEL
LIN {X 0,Y 193.289,Z 770.981,A -85,B 0,C 180,E1 4667.862,E2 4667.862} C_VEL
LIN {X 0,Y 176.523,Z 785.657,A -85,B 0,C 180,E1 4664.897,E2 4664.897} C_VEL
LIN {X 0,Y 160.417,Z 798.113,A -85,B 0,C 180,E1 4661.329,E2 4661.329} C_VEL
LIN {X 0,Y 143.028,Z 809.934,A -85,B 0,C 180,E1 4656.312,E2 4656.312} C_VEL
LIN {X 0,Y 129.191,Z 818.386,A -85,B 0,C 180,E1 4650.989,E2 4650.989} C_VEL
LIN {X 0,Y 114.122,Z 826.867,A -85,B 0,C 180,E1 4642.869,E2 4642.869} C_VEL
LIN {X 0,Y 102.297,Z 833.024,A -85,B 0,C 180,E1 4633.17,E2 4633.17} C_VEL
LIN {X 0,Y 93.754,Z 837.621,A -85,B 0,C 180,E1 4621.504,E2 4621.504} C_VEL
LIN {X 0,Y 88.952,Z 840.628,A -85,B 0,C 180,E1 4607.667,E2 4607.667} C_VEL
LIN {X 0,Y 88.02,Z 841.775,A -85,B 0,C 180,E1 4596.522,E2 4596.522} C_VEL
LIN {X 0,Y 88.05,Z 842.006,A -85,B 0,C 180,E1 4588.699,E2 4588.699} C_VEL
LIN {X 0,Y 88.16,Z 841.481,A -85,B 0,C 180,E1 4578.884,E2 4578.884} C_VEL
LIN {X 0,Y 90.592,Z 839.448,A -85,B 0,C 180,E1 4565.898,E2 4565.898} C_VEL
LIN {X 0,Y 96.192,Z 836.238,A -85,B 0,C 180,E1 4554.404,E2 4554.404} C_VEL
LIN {X 0,Y 105.411,Z 831.469,A -85,B 0,C 180,E1 4543.823,E2 4543.823} C_VEL
LIN {X 0,Y 108.638,Z 829.415,A -85,B 0,C 180,E1 4540.209,E2 4540.209} C_VEL
LIN {X 0,Y 116.011,Z 823.409,A -85,B 0,C 180,E1 4530.49,E2 4530.49} C_VEL
LIN {X 0,Y 119.872,Z 821.175,A -85,B 0,C 180,E1 4528.08,E2 4528.08} C_VEL
LIN {X 0,Y 136.589,Z 811.676,A -85,B 0,C 180,E1 4521.621,E2 4521.621} C_VEL
LIN {X 0,Y 152.202,Z 801.801,A -85,B 0,C 180,E1 4517.195,E2 4517.195} C_VEL
LIN {X 0,Y 170.603,Z 788.52,A -85,B 0,C 180,E1 4513.213,E2 4513.213} C_VEL
LIN {X 0,Y 186.125,Z 775.714,A -85,B 0,C 180,E1 4510.567,E2 4510.567} C_VEL
LIN {X 0,Y 203.52,Z 759.332,A -85,B 0,C 180,E1 4508.149,E2 4508.149} C_VEL
LIN {X 0,Y 218.341,Z 743.175,A -85,B 0,C 180,E1 4506.44,E2 4506.44} C_VEL
LIN {X 0,Y 232.849,Z 724.921,A -85,B 0,C 180,E1 4505.007,E2 4505.007} C_VEL
LIN {X 0,Y 244.8,Z 707.408,A -85,B 0,C 180,E1 4503.981,E2 4503.981} C_VEL
LIN {X 0,Y 255.826,Z 688.612,A -85,B 0,C 180,E1 4503.137,E2 4503.137} C_VEL
LIN {X 0,Y 265.699,Z 668.471,A -85,B 0,C 180,E1 4502.454,E2 4502.454} C_VEL
LIN {X 0,Y 274.109,Z 647.649,A -85,B 0,C 180,E1 4501.93,E2 4501.93} C_VEL
LIN {X 0,Y 281.332,Z 624.561,A -85,B 0,C 180,E1 4501.514,E2 4501.514} C_VEL
LIN {X 0,Y 286.462,Z 602.197,A -85,B 0,C 180,E1 4501.177,E2 4501.177} C_VEL
LIN {X 0,Y 290.822,Z 571.474,A -85,B 0,C 180,E1 4500.745,E2 4500.745} C_VEL
LIN {X 0,Y 294.39,Z 542.194,A -85,B 0,C 180,E1 4500.341,E2 4500.341} C_VEL
LIN {X 0,Y 294.617,Z 542.889,A -85,B 0,C 180,E1 4497.082,E2 4497.082} C_VEL
LIN {X 0,Y 294.904,Z 543.918,A -85,B 0,C 180,E1 4495.722,E2 4495.722} C_VEL
LIN {X 0,Y 295.656,Z 546.699,A -85,B 0,C 180,E1 4493.397,E2 4493.397} C_VEL
LIN {X 0,Y 301.661,Z 557.666,A -85,B 0,C 180,E1 4485.606,E2 4485.606} C_VEL
LIN {X 0,Y 306.516,Z 561.968,A -85,B 0,C 180,E1 4482.046,E2 4482.046} C_VEL
LIN {X 0,Y 312.738,Z 566.776,A -85,B 0,C 180,E1 4478.231,E2 4478.231} C_VEL
LIN {X 0,Y 317.28,Z 569.524,A -85,B 0,C 180,E1 4475.22,E2 4475.22} C_VEL
LIN {X 0,Y 319.6,Z 571.363,A -85,B 0,C 180,E1 4473.525,E2 4473.525} C_VEL
LIN {X 0,Y 323.018,Z 574.38,A -85,B 0,C 180,E1 4470.721,E2 4470.721} C_VEL
LIN {X 0,Y 326.714,Z 577.145,A -85,B 0,C 180,E1 4467.307,E2 4467.307} C_VEL
LIN {X 0,Y 328.261,Z 578.555,A -85,B 0,C 180,E1 4465.702,E2 4465.702} C_VEL
LIN {X 0,Y 331.614,Z 582.166,A -85,B 0,C 180,E1 4462.042,E2 4462.042} C_VEL
LIN {X 0,Y 335.081,Z 584.751,A -85,B 0,C 180,E1 4458.286,E2 4458.286} C_VEL
LIN {X 0,Y 336.503,Z 586.038,A -85,B 0,C 180,E1 4456.656,E2 4456.656} C_VEL
LIN {X 0,Y 339.647,Z 589.503,A -85,B 0,C 180,E1 4452.844,E2 4452.844} C_VEL
LIN {X 0,Y 342.658,Z 591.811,A -85,B 0,C 180,E1 4449.069,E2 4449.069} C_VEL
LIN {X 0,Y 344.948,Z 593.325,A -85,B 0,C 180,E1 4446.031,E2 4446.031} C_VEL
LIN {X 0,Y 347.36,Z 596.368,A -85,B 0,C 180,E1 4442.369,E2 4442.369} C_VEL
LIN {X 0,Y 349.702,Z 598.443,A -85,B 0,C 180,E1 4438.626,E2 4438.626} C_VEL
LIN {X 0,Y 351.87,Z 599.753,A -85,B 0,C 180,E1 4434.869,E2 4434.869} C_VEL
LIN {X 0,Y 353.791,Z 600.61,A -85,B 0,C 180,E1 4431.153,E2 4431.153} C_VEL
LIN {X 0,Y 355.139,Z 602.661,A -85,B 0,C 180,E1 4427.532,E2 4427.532} C_VEL
LIN {X 0,Y 356.361,Z 604.186,A -85,B 0,C 180,E1 4423.963,E2 4423.963} C_VEL
LIN {X 0,Y 357.21,Z 605.149,A -85,B 0,C 180,E1 4420.482,E2 4420.482} C_VEL
LIN {X 0,Y 357.95,Z 605.732,A -85,B 0,C 180,E1 4416.898,E2 4416.898} C_VEL
LIN {X 0,Y 358.281,Z 606.03,A -85,B 0,C 180,E1 4413.52,E2 4413.52} C_VEL
LIN {X 0,Y 358.499,Z 606.154,A -85,B 0,C 180,E1 4410,E2 4410} C_VEL
LIN {X 0,Y 358.282,Z 606.03,A -85,B 0,C 180,E1 4406.48,E2 4406.48} C_VEL
LIN {X 0,Y 357.946,Z 605.706,A -85,B 0,C 180,E1 4402.94,E2 4402.94} C_VEL
LIN {X 0,Y 357.158,Z 605.102,A -85,B 0,C 180,E1 4399.301,E2 4399.301} C_VEL
LIN {X 0,Y 356.261,Z 604.059,A -85,B 0,C 180,E1 4395.702,E2 4395.702} C_VEL
LIN {X 0,Y 355.078,Z 602.579,A -85,B 0,C 180,E1 4392.296,E2 4392.296} C_VEL
LIN {X 0,Y 353.659,Z 600.534,A -85,B 0,C 180,E1 4388.611,E2 4388.611} C_VEL
LIN {X 0,Y 351.775,Z 599.701,A -85,B 0,C 180,E1 4384.945,E2 4384.945} C_VEL
LIN {X 0,Y 349.538,Z 598.32,A -85,B 0,C 180,E1 4381.082,E2 4381.082} C_VEL
LIN {X 0,Y 347.223,Z 596.226,A -85,B 0,C 180,E1 4377.421,E2 4377.421} C_VEL
LIN {X 0,Y 344.707,Z 592.997,A -85,B 0,C 180,E1 4373.631,E2 4373.631} C_VEL
LIN {X 0,Y 341.675,Z 591.162,A -85,B 0,C 180,E1 4369.706,E2 4369.706} C_VEL
LIN {X 0,Y 338.727,Z 588.616,A -85,B 0,C 180,E1 4366.074,E2 4366.074} C_VEL
LIN {X 0,Y 335.423,Z 584.942,A -85,B 0,C 180,E1 4362.079,E2 4362.079} C_VEL
LIN {X 0,Y 331.981,Z 582.48,A -85,B 0,C 180,E1 4358.347,E2 4358.347} C_VEL
LIN {X 0,Y 328.521,Z 578.896,A -85,B 0,C 180,E1 4354.584,E2 4354.584} C_VEL
LIN {X 0,Y 326.992,Z 577.325,A -85,B 0,C 180,E1 4352.975,E2 4352.975} C_VEL
LIN {X 0,Y 323.237,Z 574.549,A -85,B 0,C 180,E1 4349.461,E2 4349.461} C_VEL
LIN {X 0,Y 319.711,Z 571.472,A -85,B 0,C 180,E1 4346.565,E2 4346.565} C_VEL
LIN {X 0,Y 317.451,Z 569.612,A -85,B 0,C 180,E1 4344.896,E2 4344.896} C_VEL
LIN {X 0,Y 313.007,Z 566.965,A -85,B 0,C 180,E1 4341.946,E2 4341.946} C_VEL
LIN {X 0,Y 306.792,Z 562.225,A -85,B 0,C 180,E1 4338.134,E2 4338.134} C_VEL
LIN {X 0,Y 303.033,Z 558.963,A -85,B 0,C 180,E1 4335.501,E2 4335.501} C_VEL
LIN {X 0,Y 298.401,Z 553.171,A -85,B 0,C 180,E1 4331.108,E2 4331.108} C_VEL
LIN {X 0,Y 295.24,Z 545.141,A -85,B 0,C 180,E1 4325.441,E2 4325.441} C_VEL
LIN {X 0,Y 294.7,Z 543.041,A -85,B 0,C 180,E1 4323.307,E2 4323.307} C_VEL
LIN {X 0,Y 294.386,Z 542.169,A -85,B 0,C 180,E1 4319.805,E2 4319.805} C_VEL
LIN {X 0,Y 294.364,Z 542.402,A -85,B 0,C 180,E1 4319.652,E2 4319.652} C_VEL
LIN {X 0,Y 287.41,Z 596.855,A -85,B 0,C 180,E1 4318.901,E2 4318.901} C_VEL
LIN {X 0,Y 282.455,Z 620.237,A -85,B 0,C 180,E1 4318.552,E2 4318.552} C_VEL
LIN {X 0,Y 275.844,Z 642.645,A -85,B 0,C 180,E1 4318.169,E2 4318.169} C_VEL
LIN {X 0,Y 267.675,Z 663.956,A -85,B 0,C 180,E1 4317.673,E2 4317.673} C_VEL
LIN {X 0,Y 258.792,Z 682.889,A -85,B 0,C 180,E1 4317.081,E2 4317.081} C_VEL
LIN {X 0,Y 247.492,Z 703.135,A -85,B 0,C 180,E1 4316.234,E2 4316.234} C_VEL
LIN {X 0,Y 235.28,Z 721.52,A -85,B 0,C 180,E1 4315.215,E2 4315.215} C_VEL
LIN {X 0,Y 221.23,Z 739.786,A -85,B 0,C 180,E1 4313.864,E2 4313.864} C_VEL
LIN {X 0,Y 206.848,Z 755.863,A -85,B 0,C 180,E1 4312.264,E2 4312.264} C_VEL
LIN {X 0,Y 191.729,Z 770.726,A -85,B 0,C 180,E1 4310.265,E2 4310.265} C_VEL
LIN {X 0,Y 175.055,Z 785.013,A -85,B 0,C 180,E1 4307.6,E2 4307.6} C_VEL
LIN {X 0,Y 157.964,Z 797.86,A -85,B 0,C 180,E1 4304.171,E2 4304.171} C_VEL
LIN {X 0,Y 139.904,Z 809.678,A -85,B 0,C 180,E1 4299.422,E2 4299.422} C_VEL
LIN {X 0,Y 125.378,Z 818.13,A -85,B 0,C 180,E1 4294.305,E2 4294.305} C_VEL
LIN {X 0,Y 109.317,Z 826.607,A -85,B 0,C 180,E1 4286.335,E2 4286.335} C_VEL
LIN {X 0,Y 96.43,Z 832.77,A -85,B 0,C 180,E1 4276.535,E2 4276.535} C_VEL
LIN {X 0,Y 86.843,Z 837.366,A -85,B 0,C 180,E1 4264.342,E2 4264.342} C_VEL
LIN {X 0,Y 81.224,Z 840.376,A -85,B 0,C 180,E1 4249.412,E2 4249.412} C_VEL
LIN {X 0,Y 80.032,Z 841.526,A -85,B 0,C 180,E1 4237.177,E2 4237.177} C_VEL
LIN {X 0,Y 80.05,Z 841.757,A -85,B 0,C 180,E1 4228.569,E2 4228.569} C_VEL
LIN {X 0,Y 80.231,Z 841.228,A -85,B 0,C 180,E1 4217.769,E2 4217.769} C_VEL
LIN {X 0,Y 83.181,Z 839.195,A -85,B 0,C 180,E1 4203.593,E2 4203.593} C_VEL
LIN {X 0,Y 89.613,Z 835.984,A -85,B 0,C 180,E1 4191.332,E2 4191.332} C_VEL
LIN {X 0,Y 101.417,Z 830.468,A -85,B 0,C 180,E1 4179.121,E2 4179.121} C_VEL
LIN {X 0,Y 115.807,Z 823.257,A -85,B 0,C 180,E1 4170.05,E2 4170.05} C_VEL
LIN {X 0,Y 119.872,Z 821.175,A -85,B 0,C 180,E1 4168.08,E2 4168.08} C_VEL
LIN {X 0,Y 124.497,Z 818.453,A -85,B 0,C 180,E1 4165.447,E2 4165.447} C_VEL
LIN {X 0,Y 135.489,Z 810.634,A -85,B 0,C 180,E1 4158.2,E2 4158.2} C_VEL
LIN {X 0,Y 140.06,Z 807.789,A -85,B 0,C 180,E1 4156.571,E2 4156.571} C_VEL
LIN {X 0,Y 157.736,Z 796.326,A -85,B 0,C 180,E1 4152.539,E2 4152.539} C_VEL
LIN {X 0,Y 174.614,Z 783.878,A -85,B 0,C 180,E1 4149.559,E2 4149.559} C_VEL
LIN {X 0,Y 192.422,Z 768.699,A -85,B 0,C 180,E1 4147.05,E2 4147.05} C_VEL
LIN {X 0,Y 207.359,Z 754.122,A -85,B 0,C 180,E1 4145.321,E2 4145.321} C_VEL
LIN {X 0,Y 222.953,Z 736.596,A -85,B 0,C 180,E1 4143.803,E2 4143.803} C_VEL
LIN {X 0,Y 236.22,Z 719.21,A -85,B 0,C 180,E1 4142.689,E2 4142.689} C_VEL
LIN {X 0,Y 249.074,Z 699.633,A -85,B 0,C 180,E1 4141.751,E2 4141.751} C_VEL
LIN {X 0,Y 259.501,Z 680.669,A -85,B 0,C 180,E1 4141.066,E2 4141.066} C_VEL
LIN {X 0,Y 268.466,Z 661.448,A -85,B 0,C 180,E1 4140.544,E2 4140.544} C_VEL
LIN {X 0,Y 276.703,Z 639.421,A -85,B 0,C 180,E1 4140.109,E2 4140.109} C_VEL
LIN {X 0,Y 283.235,Z 616.665,A -85,B 0,C 180,E1 4139.772,E2 4139.772} C_VEL
LIN {X 0,Y 287.938,Z 592.989,A -85,B 0,C 180,E1 4139.449,E2 4139.449} C_VEL
LIN {X 0,Y 293.426,Z 550.222,A -85,B 0,C 180,E1 4138.882,E2 4138.882} C_VEL
LIN {X 0,Y 293.79,Z 551.396,A -85,B 0,C 180,E1 4136.293,E2 4136.293} C_VEL
LIN {X 0,Y 294.501,Z 554.392,A -85,B 0,C 180,E1 4133.763,E2 4133.763} C_VEL
LIN {X 0,Y 300.262,Z 565.358,A -85,B 0,C 180,E1 4125.931,E2 4125.931} C_VEL
LIN {X 0,Y 305.148,Z 569.787,A -85,B 0,C 180,E1 4122.258,E2 4122.258} C_VEL
LIN {X 0,Y 311.53,Z 574.683,A -85,B 0,C 180,E1 4118.34,E2 4118.34} C_VEL
LIN {X 0,Y 316.092,Z 577.418,A -85,B 0,C 180,E1 4115.321,E2 4115.321} C_VEL
LIN {X 0,Y 319.699,Z 580.459,A -85,B 0,C 180,E1 4112.63,E2 4112.63} C_VEL
LIN {X 0,Y 323.399,Z 583.446,A -85,B 0,C 180,E1 4109.533,E2 4109.533} C_VEL
LIN {X 0,Y 326.912,Z 586.186,A -85,B 0,C 180,E1 4106.07,E2 4106.07} C_VEL
LIN {X 0,Y 330.215,Z 589.791,A -85,B 0,C 180,E1 4102.494,E2 4102.494} C_VEL
LIN {X 0,Y 333.83,Z 592.564,A -85,B 0,C 180,E1 4098.554,E2 4098.554} C_VEL
LIN {X 0,Y 335.362,Z 593.9,A -85,B 0,C 180,E1 4096.824,E2 4096.824} C_VEL
LIN {X 0,Y 338.412,Z 597.265,A -85,B 0,C 180,E1 4093.133,E2 4093.133} C_VEL
LIN {X 0,Y 341.442,Z 599.617,A -85,B 0,C 180,E1 4089.369,E2 4089.369} C_VEL
LIN {X 0,Y 343.849,Z 601.204,A -85,B 0,C 180,E1 4086.177,E2 4086.177} C_VEL
LIN {X 0,Y 346.298,Z 604.269,A -85,B 0,C 180,E1 4082.481,E2 4082.481} C_VEL
LIN {X 0,Y 348.728,Z 606.401,A -85,B 0,C 180,E1 4078.607,E2 4078.607} C_VEL
LIN {X 0,Y 350.854,Z 607.676,A -85,B 0,C 180,E1 4074.945,E2 4074.945} C_VEL
LIN {X 0,Y 352.791,Z 608.549,A -85,B 0,C 180,E1 4071.184,E2 4071.184} C_VEL
LIN {X 0,Y 354.142,Z 610.596,A -85,B 0,C 180,E1 4067.583,E2 4067.583} C_VEL
LIN {X 0,Y 355.336,Z 612.061,A -85,B 0,C 180,E1 4064.17,E2 4064.17} C_VEL
LIN {X 0,Y 356.187,Z 613.051,A -85,B 0,C 180,E1 4060.677,E2 4060.677} C_VEL
LIN {X 0,Y 356.968,Z 613.645,A -85,B 0,C 180,E1 4057.079,E2 4057.079} C_VEL
LIN {X 0,Y 357.305,Z 613.97,A -85,B 0,C 180,E1 4053.529,E2 4053.529} C_VEL
LIN {X 0,Y 357.524,Z 614.094,A -85,B 0,C 180,E1 4050,E2 4050} C_VEL
LIN {X 0,Y 357.305,Z 613.971,A -85,B 0,C 180,E1 4046.471,E2 4046.471} C_VEL
LIN {X 0,Y 356.968,Z 613.645,A -85,B 0,C 180,E1 4042.921,E2 4042.921} C_VEL
LIN {X 0,Y 356.174,Z 613.039,A -85,B 0,C 180,E1 4039.272,E2 4039.272} C_VEL
LIN {X 0,Y 355.266,Z 611.995,A -85,B 0,C 180,E1 4035.661,E2 4035.661} C_VEL
LIN {X 0,Y 354.082,Z 610.513,A -85,B 0,C 180,E1 4032.244,E2 4032.244} C_VEL
LIN {X 0,Y 352.642,Z 608.463,A -85,B 0,C 180,E1 4028.546,E2 4028.546} C_VEL
LIN {X 0,Y 350.76,Z 607.625,A -85,B 0,C 180,E1 4024.867,E2 4024.867} C_VEL
LIN {X 0,Y 348.508,Z 606.237,A -85,B 0,C 180,E1 4020.998,E2 4020.998} C_VEL
LIN {X 0,Y 346.103,Z 604.059,A -85,B 0,C 180,E1 4017.211,E2 4017.211} C_VEL
LIN {X 0,Y 343.581,Z 600.831,A -85,B 0,C 180,E1 4013.436,E2 4013.436} C_VEL
LIN {X 0,Y 340.704,Z 599.136,A -85,B 0,C 180,E1 4009.731,E2 4009.731} C_VEL
LIN {X 0,Y 337.685,Z 596.563,A -85,B 0,C 180,E1 4006.013,E2 4006.013} C_VEL
LIN {X 0,Y 334.407,Z 592.882,A -85,B 0,C 180,E1 4002.047,E2 4002.047} C_VEL
LIN {X 0,Y 331.101,Z 590.563,A -85,B 0,C 180,E1 3998.468,E2 3998.468} C_VEL
LIN {X 0,Y 327.616,Z 587.078,A -85,B 0,C 180,E1 3994.693,E2 3994.693} C_VEL
LIN {X 0,Y 325.793,Z 585.161,A -85,B 0,C 180,E1 3992.767,E2 3992.767} C_VEL
LIN {X 0,Y 322.355,Z 582.641,A -85,B 0,C 180,E1 3989.549,E2 3989.549} C_VEL
LIN {X 0,Y 318.728,Z 579.594,A -85,B 0,C 180,E1 3986.616,E2 3986.616} C_VEL
LIN {X 0,Y 316.092,Z 577.418,A -85,B 0,C 180,E1 3984.679,E2 3984.679} C_VEL
LIN {X 0,Y 311.53,Z 574.683,A -85,B 0,C 180,E1 3981.66,E2 3981.66} C_VEL
LIN {X 0,Y 304.879,Z 569.527,A -85,B 0,C 180,E1 3977.561,E2 3977.561} C_VEL
LIN {X 0,Y 297.643,Z 561.853,A -85,B 0,C 180,E1 3971.431,E2 3971.431} C_VEL
LIN {X 0,Y 294.169,Z 552.99,A -85,B 0,C 180,E1 3965.218,E2 3965.218} C_VEL
LIN {X 0,Y 293.641,Z 550.853,A -85,B 0,C 180,E1 3962.928,E2 3962.928} C_VEL
LIN {X 0,Y 293.401,Z 550.418,A -85,B 0,C 180,E1 3961.108,E2 3961.108} C_VEL
LIN {X 0,Y 287.248,Z 597.36,A -85,B 0,C 180,E1 3960.492,E2 3960.492} C_VEL
LIN {X 0,Y 282.235,Z 620.498,A -85,B 0,C 180,E1 3960.175,E2 3960.175} C_VEL
LIN {X 0,Y 275.454,Z 643.104,A -85,B 0,C 180,E1 3959.827,E2 3959.827} C_VEL
LIN {X 0,Y 267.469,Z 663.711,A -85,B 0,C 180,E1 3959.399,E2 3959.399} C_VEL
LIN {X 0,Y 258.507,Z 682.64,A -85,B 0,C 180,E1 3958.871,E2 3958.871} C_VEL
LIN {X 0,Y 247.092,Z 702.88,A -85,B 0,C 180,E1 3958.111,E2 3958.111} C_VEL
LIN {X 0,Y 234.741,Z 721.271,A -85,B 0,C 180,E1 3957.194,E2 3957.194} C_VEL
LIN {X 0,Y 220.507,Z 739.531,A -85,B 0,C 180,E1 3955.975,E2 3955.975} C_VEL
LIN {X 0,Y 205.421,Z 756.109,A -85,B 0,C 180,E1 3954.471,E2 3954.471} C_VEL
LIN {X 0,Y 189.556,Z 771.356,A -85,B 0,C 180,E1 3952.577,E2 3952.577} C_VEL
LIN {X 0,Y 172.535,Z 785.478,A -85,B 0,C 180,E1 3950.11,E2 3950.11} C_VEL
LIN {X 0,Y 155.003,Z 798.225,A -85,B 0,C 180,E1 3946.908,E2 3946.908} C_VEL
LIN {X 0,Y 136.873,Z 809.616,A -85,B 0,C 180,E1 3942.572,E2 3942.572} C_VEL
LIN {X 0,Y 121.195,Z 818.309,A -85,B 0,C 180,E1 3937.514,E2 3937.514} C_VEL
LIN {X 0,Y 104.223,Z 826.682,A -85,B 0,C 180,E1 3929.699,E2 3929.699} C_VEL
LIN {X 0,Y 90.342,Z 832.77,A -85,B 0,C 180,E1 3919.786,E2 3919.786} C_VEL
LIN {X 0,Y 79.314,Z 837.493,A -85,B 0,C 180,E1 3906.215,E2 3906.215} C_VEL
LIN {X 0,Y 73.245,Z 840.298,A -85,B 0,C 180,E1 3889.954,E2 3889.954} C_VEL
LIN {X 0,Y 72.034,Z 841.307,A -85,B 0,C 180,E1 3877.176,E2 3877.176} C_VEL
LIN {X 0,Y 72.051,Z 841.508,A -85,B 0,C 180,E1 3868.41,E2 3868.41} C_VEL
LIN {X 0,Y 72.262,Z 841.054,A -85,B 0,C 180,E1 3857.21,E2 3857.21} C_VEL
LIN {X 0,Y 75.641,Z 839.085,A -85,B 0,C 180,E1 3841.585,E2 3841.585} C_VEL
LIN {X 0,Y 83.331,Z 835.731,A -85,B 0,C 180,E1 3827.786,E2 3827.786} C_VEL
LIN {X 0,Y 95.949,Z 830.404,A -85,B 0,C 180,E1 3815.63,E2 3815.63} C_VEL
LIN {X 0,Y 111.685,Z 823.098,A -85,B 0,C 180,E1 3806.463,E2 3806.463} C_VEL
LIN {X 0,Y 128.654,Z 814.376,A -85,B 0,C 180,E1 3799.89,E2 3799.89} C_VEL
LIN {X 0,Y 140.06,Z 807.789,A -85,B 0,C 180,E1 3796.571,E2 3796.571} C_VEL
LIN {X 0,Y 145.415,Z 804.374,A -85,B 0,C 180,E1 3794.774,E2 3794.774} C_VEL
LIN {X 0,Y 157.54,Z 795.366,A -85,B 0,C 180,E1 3789.733,E2 3789.733} C_VEL
LIN {X 0,Y 163.053,Z 791.331,A -85,B 0,C 180,E1 3788.418,E2 3788.418} C_VEL
LIN {X 0,Y 180.921,Z 777.613,A -85,B 0,C 180,E1 3785.879,E2 3785.879} C_VEL
LIN {X 0,Y 196.469,Z 763.98,A -85,B 0,C 180,E1 3784.086,E2 3784.086} C_VEL
LIN {X 0,Y 213.165,Z 747.097,A -85,B 0,C 180,E1 3782.49,E2 3782.49} C_VEL
LIN {X 0,Y 227.026,Z 730.802,A -85,B 0,C 180,E1 3781.363,E2 3781.363} C_VEL
LIN {X 0,Y 240.965,Z 711.842,A -85,B 0,C 180,E1 3780.389,E2 3780.389} C_VEL
LIN {X 0,Y 252.962,Z 692.529,A -85,B 0,C 180,E1 3779.651,E2 3779.651} C_VEL
LIN {X 0,Y 263.489,Z 672.39,A -85,B 0,C 180,E1 3779.076,E2 3779.076} C_VEL
LIN {X 0,Y 272.029,Z 652.445,A -85,B 0,C 180,E1 3778.654,E2 3778.654} C_VEL
LIN {X 0,Y 279.478,Z 630.642,A -85,B 0,C 180,E1 3778.324,E2 3778.324} C_VEL
LIN {X 0,Y 285.274,Z 608.04,A -85,B 0,C 180,E1 3778.042,E2 3778.042} C_VEL
LIN {X 0,Y 288.97,Z 586.871,A -85,B 0,C 180,E1 3777.778,E2 3777.778} C_VEL
LIN {X 0,Y 292.603,Z 558.684,A -85,B 0,C 180,E1 3777.405,E2 3777.405} C_VEL
LIN {X 0,Y 292.917,Z 560.146,A -85,B 0,C 180,E1 3775.693,E2 3775.693} C_VEL
LIN {X 0,Y 295.149,Z 567.074,A -85,B 0,C 180,E1 3770.543,E2 3770.543} C_VEL
LIN {X 0,Y 299.08,Z 573.276,A -85,B 0,C 180,E1 3766.072,E2 3766.072} C_VEL
LIN {X 0,Y 303.919,Z 577.729,A -85,B 0,C 180,E1 3762.382,E2 3762.382} C_VEL
LIN {X 0,Y 310.585,Z 582.774,A -85,B 0,C 180,E1 3758.271,E2 3758.271} C_VEL
LIN {X 0,Y 315.461,Z 585.58,A -85,B 0,C 180,E1 3755.068,E2 3755.068} C_VEL
LIN {X 0,Y 319.65,Z 589.343,A -85,B 0,C 180,E1 3751.815,E2 3751.815} C_VEL
LIN {X 0,Y 323.634,Z 592.387,A -85,B 0,C 180,E1 3748.318,E2 3748.318} C_VEL
LIN {X 0,Y 325.826,Z 594.159,A -85,B 0,C 180,E1 3746.154,E2 3746.154} C_VEL
LIN {X 0,Y 329.14,Z 597.711,A -85,B 0,C 180,E1 3742.587,E2 3742.587} C_VEL
LIN {X 0,Y 332.773,Z 600.485,A -85,B 0,C 180,E1 3738.623,E2 3738.623} C_VEL
LIN {X 0,Y 334.212,Z 601.761,A -85,B 0,C 180,E1 3736.992,E2 3736.992} C_VEL
LIN {X 0,Y 337.178,Z 605.038,A -85,B 0,C 180,E1 3733.405,E2 3733.405} C_VEL
LIN {X 0,Y 340.255,Z 607.447,A -85,B 0,C 180,E1 3729.617,E2 3729.617} C_VEL
LIN {X 0,Y 342.761,Z 609.096,A -85,B 0,C 180,E1 3726.31,E2 3726.31} C_VEL
LIN {X 0,Y 345.253,Z 612.185,A -85,B 0,C 180,E1 3722.57,E2 3722.57} C_VEL
LIN {X 0,Y 347.58,Z 614.233,A -85,B 0,C 180,E1 3718.899,E2 3718.899} C_VEL
LIN {X 0,Y 349.745,Z 615.549,A -85,B 0,C 180,E1 3715.211,E2 3715.211} C_VEL
LIN {X 0,Y 351.626,Z 616.391,A -85,B 0,C 180,E1 3711.519,E2 3711.519} C_VEL
LIN {X 0,Y 353.085,Z 618.449,A -85,B 0,C 180,E1 3707.808,E2 3707.808} C_VEL
LIN {X 0,Y 354.27,Z 619.93,A -85,B 0,C 180,E1 3704.38,E2 3704.38} C_VEL
LIN {X 0,Y 355.203,Z 620.988,A -85,B 0,C 180,E1 3700.706,E2 3700.706} C_VEL
LIN {X 0,Y 355.99,Z 621.585,A -85,B 0,C 180,E1 3697.099,E2 3697.099} C_VEL
LIN {X 0,Y 356.329,Z 621.91,A -85,B 0,C 180,E1 3693.539,E2 3693.539} C_VEL
LIN {X 0,Y 356.549,Z 622.034,A -85,B 0,C 180,E1 3690,E2 3690} C_VEL
LIN {X 0,Y 356.329,Z 621.911,A -85,B 0,C 180,E1 3686.461,E2 3686.461} C_VEL
LIN {X 0,Y 355.99,Z 621.585,A -85,B 0,C 180,E1 3682.901,E2 3682.901} C_VEL
LIN {X 0,Y 355.202,Z 620.988,A -85,B 0,C 180,E1 3679.294,E2 3679.294} C_VEL
LIN {X 0,Y 354.27,Z 619.93,A -85,B 0,C 180,E1 3675.62,E2 3675.62} C_VEL
LIN {X 0,Y 353.086,Z 618.448,A -85,B 0,C 180,E1 3672.192,E2 3672.192} C_VEL
LIN {X 0,Y 351.626,Z 616.391,A -85,B 0,C 180,E1 3668.481,E2 3668.481} C_VEL
LIN {X 0,Y 349.746,Z 615.549,A -85,B 0,C 180,E1 3664.789,E2 3664.789} C_VEL
LIN {X 0,Y 347.474,Z 614.15,A -85,B 0,C 180,E1 3660.903,E2 3660.903} C_VEL
LIN {X 0,Y 345.088,Z 612.008,A -85,B 0,C 180,E1 3657.166,E2 3657.166} C_VEL
LIN {X 0,Y 342.606,Z 608.881,A -85,B 0,C 180,E1 3653.463,E2 3653.463} C_VEL
LIN {X 0,Y 339.64,Z 607.045,A -85,B 0,C 180,E1 3649.636,E2 3649.636} C_VEL
LIN {X 0,Y 336.644,Z 604.509,A -85,B 0,C 180,E1 3645.952,E2 3645.952} C_VEL
LIN {X 0,Y 333.319,Z 600.781,A -85,B 0,C 180,E1 3641.935,E2 3641.935} C_VEL
LIN {X 0,Y 329.846,Z 598.34,A -85,B 0,C 180,E1 3638.198,E2 3638.198} C_VEL
LIN {X 0,Y 326.445,Z 594.933,A -85,B 0,C 180,E1 3634.516,E2 3634.516} C_VEL
LIN {X 0,Y 324.616,Z 593.03,A -85,B 0,C 180,E1 3632.617,E2 3632.617} C_VEL
LIN {X 0,Y 320.948,Z 590.385,A -85,B 0,C 180,E1 3629.277,E2 3629.277} C_VEL
LIN {X 0,Y 316.904,Z 586.923,A -85,B 0,C 180,E1 3626.012,E2 3626.012} C_VEL
LIN {X 0,Y 314.671,Z 585.18,A -85,B 0,C 180,E1 3624.398,E2 3624.398} C_VEL
LIN {X 0,Y 309.394,Z 581.999,A -85,B 0,C 180,E1 3621.021,E2 3621.021} C_VEL
LIN {X 0,Y 300.29,Z 574.463,A -85,B 0,C 180,E1 3614.954,E2 3614.954} C_VEL
LIN {X 0,Y 295.743,Z 568.413,A -85,B 0,C 180,E1 3610.322,E2 3610.322} C_VEL
LIN {X 0,Y 292.965,Z 560.347,A -85,B 0,C 180,E1 3604.502,E2 3604.502} C_VEL
LIN {X 0,Y 292.611,Z 558.703,A -85,B 0,C 180,E1 3602.644,E2 3602.644} C_VEL
LIN {X 0,Y 292.556,Z 559.013,A -85,B 0,C 180,E1 3602.567,E2 3602.567} C_VEL
LIN {X 0,Y 287.274,Z 598.01,A -85,B 0,C 180,E1 3602.083,E2 3602.083} C_VEL
LIN {X 0,Y 282.216,Z 620.857,A -85,B 0,C 180,E1 3601.797,E2 3601.797} C_VEL
LIN {X 0,Y 275.548,Z 642.847,A -85,B 0,C 180,E1 3601.5,E2 3601.5} C_VEL
LIN {X 0,Y 267.506,Z 663.467,A -85,B 0,C 180,E1 3601.127,E2 3601.127} C_VEL
LIN {X 0,Y 258.508,Z 682.324,A -85,B 0,C 180,E1 3600.665,E2 3600.665} C_VEL
LIN {X 0,Y 246.958,Z 702.625,A -85,B 0,C 180,E1 3599.992,E2 3599.992} C_VEL
LIN {X 0,Y 234.271,Z 721.317,A -85,B 0,C 180,E1 3599.165,E2 3599.165} C_VEL
LIN {X 0,Y 219.8,Z 739.603,A -85,B 0,C 180,E1 3598.072,E2 3598.072} C_VEL
LIN {X 0,Y 204.794,Z 755.859,A -85,B 0,C 180,E1 3596.753,E2 3596.753} C_VEL
LIN {X 0,Y 188.67,Z 771.101,A -85,B 0,C 180,E1 3595.054,E2 3595.054} C_VEL
LIN {X 0,Y 171.311,Z 785.225,A -85,B 0,C 180,E1 3592.828,E2 3592.828} C_VEL
LIN {X 0,Y 153.342,Z 797.967,A -85,B 0,C 180,E1 3589.918,E2 3589.918} C_VEL
LIN {X 0,Y 134.973,Z 809.166,A -85,B 0,C 180,E1 3586.025,E2 3586.025} C_VEL
LIN {X 0,Y 118.271,Z 818.053,A -85,B 0,C 180,E1 3581.229,E2 3581.229} C_VEL
LIN {X 0,Y 100.294,Z 826.422,A -85,B 0,C 180,E1 3573.794,E2 3573.794} C_VEL
LIN {X 0,Y 85.231,Z 832.516,A -85,B 0,C 180,E1 3564.04,E2 3564.04} C_VEL
LIN {X 0,Y 72.894,Z 837.212,A -85,B 0,C 180,E1 3550.141,E2 3550.141} C_VEL
LIN {X 0,Y 65.638,Z 840.046,A -85,B 0,C 180,E1 3532.384,E2 3532.384} C_VEL
LIN {X 0,Y 64.053,Z 841.057,A -85,B 0,C 180,E1 3518.076,E2 3518.076} C_VEL
LIN {X 0,Y 64.05,Z 841.26,A -85,B 0,C 180,E1 3508.211,E2 3508.211} C_VEL
LIN {X 0,Y 64.383,Z 840.802,A -85,B 0,C 180,E1 3495.613,E2 3495.613} C_VEL
LIN {X 0,Y 68.54,Z 838.832,A -85,B 0,C 180,E1 3478.321,E2 3478.321} C_VEL
LIN {X 0,Y 77.418,Z 835.477,A -85,B 0,C 180,E1 3463.679,E2 3463.679} C_VEL
LIN {X 0,Y 92.084,Z 829.863,A -85,B 0,C 180,E1 3450.934,E2 3450.934} C_VEL
LIN {X 0,Y 109.059,Z 822.47,A -85,B 0,C 180,E1 3442.189,E2 3442.189} C_VEL
LIN {X 0,Y 126.955,Z 813.65,A -85,B 0,C 180,E1 3436.094,E2 3436.094} C_VEL
LIN {X 0,Y 144.994,Z 803.236,A -85,B 0,C 180,E1 3431.71,E2 3431.71} C_VEL
LIN {X 0,Y 163.053,Z 791.331,A -85,B 0,C 180,E1 3428.418,E2 3428.418} C_VEL
LIN {X 0,Y 168.581,Z 787.184,A -85,B 0,C 180,E1 3427.202,E2 3427.202} C_VEL
LIN {X 0,Y 181.361,Z 776.547,A -85,B 0,C 180,E1 3423.487,E2 3423.487} C_VEL
LIN {X 0,Y 186.885,Z 771.926,A -85,B 0,C 180,E1 3422.579,E2 3422.579} C_VEL
LIN {X 0,Y 203.499,Z 756.602,A -85,B 0,C 180,E1 3421.039,E2 3421.039} C_VEL
LIN {X 0,Y 218.964,Z 740.161,A -85,B 0,C 180,E1 3419.85,E2 3419.85} C_VEL
LIN {X 0,Y 234.006,Z 721.452,A -85,B 0,C 180,E1 3418.864,E2 3418.864} C_VEL
LIN {X 0,Y 247.09,Z 702.369,A -85,B 0,C 180,E1 3418.128,E2 3418.128} C_VEL
LIN {X 0,Y 258.643,Z 682.244,A -85,B 0,C 180,E1 3417.549,E2 3417.549} C_VEL
LIN {X 0,Y 267.786,Z 663.222,A -85,B 0,C 180,E1 3417.148,E2 3417.148} C_VEL
LIN {X 0,Y 276.128,Z 641.875,A -85,B 0,C 180,E1 3416.821,E2 3416.821} C_VEL
LIN {X 0,Y 283.111,Z 618.619,A -85,B 0,C 180,E1 3416.552,E2 3416.552} C_VEL
LIN {X 0,Y 288.197,Z 594.664,A -85,B 0,C 180,E1 3416.282,E2 3416.282} C_VEL
LIN {X 0,Y 291.867,Z 567.989,A -85,B 0,C 180,E1 3415.933,E2 3415.933} C_VEL
LIN {X 0,Y 294.336,Z 575.815,A -85,B 0,C 180,E1 3410.221,E2 3410.221} C_VEL
LIN {X 0,Y 298.635,Z 581.949,A -85,B 0,C 180,E1 3405.556,E2 3405.556} C_VEL
LIN {X 0,Y 302.491,Z 585.536,A -85,B 0,C 180,E1 3402.594,E2 3402.594} C_VEL
LIN {X 0,Y 308.93,Z 590.47,A -85,B 0,C 180,E1 3398.548,E2 3398.548} C_VEL
LIN {X 0,Y 313.83,Z 593.319,A -85,B 0,C 180,E1 3395.332,E2 3395.332} C_VEL
LIN {X 0,Y 318.292,Z 597.246,A -85,B 0,C 180,E1 3391.888,E2 3391.888} C_VEL
LIN {X 0,Y 322.377,Z 600.286,A -85,B 0,C 180,E1 3388.389,E2 3388.389} C_VEL
LIN {X 0,Y 324.561,Z 602.014,A -85,B 0,C 180,E1 3386.323,E2 3386.323} C_VEL
LIN {X 0,Y 328.069,Z 605.644,A -85,B 0,C 180,E1 3382.664,E2 3382.664} C_VEL
LIN {X 0,Y 331.531,Z 608.296,A -85,B 0,C 180,E1 3378.894,E2 3378.894} C_VEL
LIN {X 0,Y 332.978,Z 609.512,A -85,B 0,C 180,E1 3377.264,E2 3377.264} C_VEL
LIN {X 0,Y 336.133,Z 612.981,A -85,B 0,C 180,E1 3373.465,E2 3373.465} C_VEL
LIN {X 0,Y 339.19,Z 615.36,A -85,B 0,C 180,E1 3369.703,E2 3369.703} C_VEL
LIN {X 0,Y 341.693,Z 617.012,A -85,B 0,C 180,E1 3366.419,E2 3366.419} C_VEL
LIN {X 0,Y 344.237,Z 620.131,A -85,B 0,C 180,E1 3362.614,E2 3362.614} C_VEL
LIN {X 0,Y 346.545,Z 622.146,A -85,B 0,C 180,E1 3358.993,E2 3358.993} C_VEL
LIN {X 0,Y 348.731,Z 623.473,A -85,B 0,C 180,E1 3355.289,E2 3355.289} C_VEL
LIN {X 0,Y 350.61,Z 624.319,A -85,B 0,C 180,E1 3351.584,E2 3351.584} C_VEL
LIN {X 0,Y 352.089,Z 626.383,A -85,B 0,C 180,E1 3347.86,E2 3347.86} C_VEL
LIN {X 0,Y 353.275,Z 627.866,A -85,B 0,C 180,E1 3344.422,E2 3344.422} C_VEL
LIN {X 0,Y 354.22,Z 628.925,A -85,B 0,C 180,E1 3340.737,E2 3340.737} C_VEL
LIN {X 0,Y 355.011,Z 629.524,A -85,B 0,C 180,E1 3337.118,E2 3337.118} C_VEL
LIN {X 0,Y 355.353,Z 629.851,A -85,B 0,C 180,E1 3333.549,E2 3333.549} C_VEL
LIN {X 0,Y 355.574,Z 629.975,A -85,B 0,C 180,E1 3330,E2 3330} C_VEL
LIN {X 0,Y 355.353,Z 629.851,A -85,B 0,C 180,E1 3326.451,E2 3326.451} C_VEL
LIN {X 0,Y 355.011,Z 629.524,A -85,B 0,C 180,E1 3322.882,E2 3322.882} C_VEL
LIN {X 0,Y 354.219,Z 628.925,A -85,B 0,C 180,E1 3319.263,E2 3319.263} C_VEL
LIN {X 0,Y 353.275,Z 627.866,A -85,B 0,C 180,E1 3315.578,E2 3315.578} C_VEL
LIN {X 0,Y 352.09,Z 626.383,A -85,B 0,C 180,E1 3312.14,E2 3312.14} C_VEL
LIN {X 0,Y 350.61,Z 624.32,A -85,B 0,C 180,E1 3308.416,E2 3308.416} C_VEL
LIN {X 0,Y 348.732,Z 623.473,A -85,B 0,C 180,E1 3304.711,E2 3304.711} C_VEL
LIN {X 0,Y 346.441,Z 622.063,A -85,B 0,C 180,E1 3300.808,E2 3300.808} C_VEL
LIN {X 0,Y 344.049,Z 619.929,A -85,B 0,C 180,E1 3297.082,E2 3297.082} C_VEL
LIN {X 0,Y 341.622,Z 616.916,A -85,B 0,C 180,E1 3293.478,E2 3293.478} C_VEL
LIN {X 0,Y 338.637,Z 614.997,A -85,B 0,C 180,E1 3289.62,E2 3289.62} C_VEL
LIN {X 0,Y 335.74,Z 612.598,A -85,B 0,C 180,E1 3286.063,E2 3286.063} C_VEL
LIN {X 0,Y 332.641,Z 609.059,A -85,B 0,C 180,E1 3282.319,E2 3282.319} C_VEL
LIN {X 0,Y 329.154,Z 606.571,A -85,B 0,C 180,E1 3278.515,E2 3278.515} C_VEL
LIN {X 0,Y 325.81,Z 603.46,A -85,B 0,C 180,E1 3274.979,E2 3274.979} C_VEL
LIN {X 0,Y 323.402,Z 600.931,A -85,B 0,C 180,E1 3272.544,E2 3272.544} C_VEL
LIN {X 0,Y 319.397,Z 598.12,A -85,B 0,C 180,E1 3269.027,E2 3269.027} C_VEL
LIN {X 0,Y 315.167,Z 594.513,A -85,B 0,C 180,E1 3265.661,E2 3265.661} C_VEL
LIN {X 0,Y 312.782,Z 592.774,A -85,B 0,C 180,E1 3263.952,E2 3263.952} C_VEL
LIN {X 0,Y 307.488,Z 589.492,A -85,B 0,C 180,E1 3260.56,E2 3260.56} C_VEL
LIN {X 0,Y 298.861,Z 582.159,A -85,B 0,C 180,E1 3254.631,E2 3254.631} C_VEL
LIN {X 0,Y 294.468,Z 576.106,A -85,B 0,C 180,E1 3249.972,E2 3249.972} C_VEL
LIN {X 0,Y 291.925,Z 568.246,A -85,B 0,C 180,E1 3244.321,E2 3244.321} C_VEL
LIN {X 0,Y 291.834,Z 568.148,A -85,B 0,C 180,E1 3244.027,E2 3244.027} C_VEL
LIN {X 0,Y 287.411,Z 599.168,A -85,B 0,C 180,E1 3243.666,E2 3243.666} C_VEL
LIN {X 0,Y 282.328,Z 621.574,A -85,B 0,C 180,E1 3243.415,E2 3243.415} C_VEL
LIN {X 0,Y 275.622,Z 643.306,A -85,B 0,C 180,E1 3243.16,E2 3243.16} C_VEL
LIN {X 0,Y 267.281,Z 664.354,A -85,B 0,C 180,E1 3242.83,E2 3242.83} C_VEL
LIN {X 0,Y 257.683,Z 684.117,A -85,B 0,C 180,E1 3242.404,E2 3242.404} C_VEL
LIN {X 0,Y 245.578,Z 704.745,A -85,B 0,C 180,E1 3241.791,E2 3241.791} C_VEL
LIN {X 0,Y 233.001,Z 722.807,A -85,B 0,C 180,E1 3241.075,E2 3241.075} C_VEL
LIN {X 0,Y 217.463,Z 741.873,A -85,B 0,C 180,E1 3240.041,E2 3240.041} C_VEL
LIN {X 0,Y 201.511,Z 758.563,A -85,B 0,C 180,E1 3238.791,E2 3238.791} C_VEL
LIN {X 0,Y 183.213,Z 774.953,A -85,B 0,C 180,E1 3237.04,E2 3237.04} C_VEL
LIN {X 0,Y 166.586,Z 787.845,A -85,B 0,C 180,E1 3235.079,E2 3235.079} C_VEL
LIN {X 0,Y 147.34,Z 800.711,A -85,B 0,C 180,E1 3232.195,E2 3232.195} C_VEL
LIN {X 0,Y 129.506,Z 810.907,A -85,B 0,C 180,E1 3228.662,E2 3228.662} C_VEL
LIN {X 0,Y 110.557,Z 820.313,A -85,B 0,C 180,E1 3223.46,E2 3223.46} C_VEL
LIN {X 0,Y 92.846,Z 827.742,A -85,B 0,C 180,E1 3216.253,E2 3216.253} C_VEL
LIN {X 0,Y 76.479,Z 833.747,A -85,B 0,C 180,E1 3205.448,E2 3205.448} C_VEL
LIN {X 0,Y 63.76,Z 837.895,A -85,B 0,C 180,E1 3189.79,E2 3189.79} C_VEL
LIN {X 0,Y 57.506,Z 840.055,A -85,B 0,C 180,E1 3172.489,E2 3172.489} C_VEL
LIN {X 0,Y 56.028,Z 840.899,A -85,B 0,C 180,E1 3156.147,E2 3156.147} C_VEL
LIN {X 0,Y 56.035,Z 840.985,A -85,B 0,C 180,E1 3146.932,E2 3146.932} C_VEL
LIN {X 0,Y 56.967,Z 840.312,A -85,B 0,C 180,E1 3130.52,E2 3130.52} C_VEL
LIN {X 0,Y 62.525,Z 838.295,A -85,B 0,C 180,E1 3112.58,E2 3112.58} C_VEL
LIN {X 0,Y 74.496,Z 834.431,A -85,B 0,C 180,E1 3096.363,E2 3096.363} C_VEL
LIN {X 0,Y 91.248,Z 828.367,A -85,B 0,C 180,E1 3084.57,E2 3084.57} C_VEL
LIN {X 0,Y 107.936,Z 821.471,A -85,B 0,C 180,E1 3077.426,E2 3077.426} C_VEL
LIN {X 0,Y 127.8,Z 811.829,A -85,B 0,C 180,E1 3071.737,E2 3071.737} C_VEL
LIN {X 0,Y 144.49,Z 802.414,A -85,B 0,C 180,E1 3068.302,E2 3068.302} C_VEL
LIN {X 0,Y 162.705,Z 790.614,A -85,B 0,C 180,E1 3065.44,E2 3065.44} C_VEL
LIN {X 0,Y 180.264,Z 777.36,A -85,B 0,C 180,E1 3063.278,E2 3063.278} C_VEL
LIN {X 0,Y 186.885,Z 771.926,A -85,B 0,C 180,E1 3062.579,E2 3062.579} C_VEL
LIN {X 0,Y 192.374,Z 767.193,A -85,B 0,C 180,E1 3061.733,E2 3061.733} C_VEL
LIN {X 0,Y 205.021,Z 754.961,A -85,B 0,C 180,E1 3058.916,E2 3058.916} C_VEL
LIN {X 0,Y 210.18,Z 749.648,A -85,B 0,C 180,E1 3058.284,E2 3058.284} C_VEL
LIN {X 0,Y 225.705,Z 732.153,A -85,B 0,C 180,E1 3057.337,E2 3057.337} C_VEL
LIN {X 0,Y 239.373,Z 714.293,A -85,B 0,C 180,E1 3056.63,E2 3056.63} C_VEL
LIN {X 0,Y 252.054,Z 694.64,A -85,B 0,C 180,E1 3056.056,E2 3056.056} C_VEL
LIN {X 0,Y 262.626,Z 675.16,A -85,B 0,C 180,E1 3055.633,E2 3055.633} C_VEL
LIN {X 0,Y 271.866,Z 654.499,A -85,B 0,C 180,E1 3055.306,E2 3055.306} C_VEL
LIN {X 0,Y 279.834,Z 632.021,A -85,B 0,C 180,E1 3055.057,E2 3055.057} C_VEL
LIN {X 0,Y 286.05,Z 608.594,A -85,B 0,C 180,E1 3054.836,E2 3054.836} C_VEL
LIN {X 0,Y 289.846,Z 587.627,A -85,B 0,C 180,E1 3054.618,E2 3054.618} C_VEL
LIN {X 0,Y 291.219,Z 578.036,A -85,B 0,C 180,E1 3054.483,E2 3054.483} C_VEL
LIN {X 0,Y 296.105,Z 588.533,A -85,B 0,C 180,E1 3046.825,E2 3046.825} C_VEL
LIN {X 0,Y 300.919,Z 593.319,A -85,B 0,C 180,E1 3042.799,E2 3042.799} C_VEL
LIN {X 0,Y 307.929,Z 598.689,A -85,B 0,C 180,E1 3038.274,E2 3038.274} C_VEL
LIN {X 0,Y 313.017,Z 601.846,A -85,B 0,C 180,E1 3034.86,E2 3034.86} C_VEL
LIN {X 0,Y 317.455,Z 605.657,A -85,B 0,C 180,E1 3031.397,E2 3031.397} C_VEL
LIN {X 0,Y 321.604,Z 608.563,A -85,B 0,C 180,E1 3027.884,E2 3027.884} C_VEL
LIN {X 0,Y 323.612,Z 610.407,A -85,B 0,C 180,E1 3025.997,E2 3025.997} C_VEL
LIN {X 0,Y 327.25,Z 613.884,A -85,B 0,C 180,E1 3022.333,E2 3022.333} C_VEL
LIN {X 0,Y 330.868,Z 616.446,A -85,B 0,C 180,E1 3018.54,E2 3018.54} C_VEL
LIN {X 0,Y 334.235,Z 620.048,A -85,B 0,C 180,E1 3014.605,E2 3014.605} C_VEL
LIN {X 0,Y 337.266,Z 622.679,A -85,B 0,C 180,E1 3010.89,E2 3010.89} C_VEL
LIN {X 0,Y 340.183,Z 624.402,A -85,B 0,C 180,E1 3007.202,E2 3007.202} C_VEL
LIN {X 0,Y 342.746,Z 627.534,A -85,B 0,C 180,E1 3003.455,E2 3003.455} C_VEL
LIN {X 0,Y 345.165,Z 629.805,A -85,B 0,C 180,E1 2999.655,E2 2999.655} C_VEL
LIN {X 0,Y 347.33,Z 631.235,A -85,B 0,C 180,E1 2995.948,E2 2995.948} C_VEL
LIN {X 0,Y 349.322,Z 632.139,A -85,B 0,C 180,E1 2992.198,E2 2992.198} C_VEL
LIN {X 0,Y 350.282,Z 633.118,A -85,B 0,C 180,E1 2990.031,E2 2990.031} C_VEL
LIN {X 0,Y 351.636,Z 635.023,A -85,B 0,C 180,E1 2986.519,E2 2986.519} C_VEL
LIN {X 0,Y 352.68,Z 636.311,A -85,B 0,C 180,E1 2982.942,E2 2982.942} C_VEL
LIN {X 0,Y 353.627,Z 637.141,A -85,B 0,C 180,E1 2979.274,E2 2979.274} C_VEL
LIN {X 0,Y 354.139,Z 637.618,A -85,B 0,C 180,E1 2975.833,E2 2975.833} C_VEL
LIN {X 0,Y 354.533,Z 637.877,A -85,B 0,C 180,E1 2972.263,E2 2972.263} C_VEL
LIN {X 0,Y 354.501,Z 637.868,A -85,B 0,C 180,E1 2968.707,E2 2968.707} C_VEL
LIN {X 0,Y 354.329,Z 637.708,A -85,B 0,C 180,E1 2965.144,E2 2965.144} C_VEL
LIN {X 0,Y 353.734,Z 637.306,A -85,B 0,C 180,E1 2961.611,E2 2961.611} C_VEL
LIN {X 0,Y 352.957,Z 636.514,A -85,B 0,C 180,E1 2957.9,E2 2957.9} C_VEL
LIN {X 0,Y 351.889,Z 635.411,A -85,B 0,C 180,E1 2954.415,E2 2954.415} C_VEL
LIN {X 0,Y 350.49,Z 633.464,A -85,B 0,C 180,E1 2950.503,E2 2950.503} C_VEL
LIN {X 0,Y 349.501,Z 632.215,A -85,B 0,C 180,E1 2948.167,E2 2948.167} C_VEL
LIN {X 0,Y 347.656,Z 631.375,A -85,B 0,C 180,E1 2944.563,E2 2944.563} C_VEL
LIN {X 0,Y 345.405,Z 629.974,A -85,B 0,C 180,E1 2940.712,E2 2940.712} C_VEL
LIN {X 0,Y 342.994,Z 627.83,A -85,B 0,C 180,E1 2936.968,E2 2936.968} C_VEL
LIN {X 0,Y 340.503,Z 624.755,A -85,B 0,C 180,E1 2933.287,E2 2933.287} C_VEL
LIN {X 0,Y 337.604,Z 622.927,A -85,B 0,C 180,E1 2929.564,E2 2929.564} C_VEL
LIN {X 0,Y 334.598,Z 620.44,A -85,B 0,C 180,E1 2925.874,E2 2925.874} C_VEL
LIN {X 0,Y 331.591,Z 617.039,A -85,B 0,C 180,E1 2922.254,E2 2922.254} C_VEL
LIN {X 0,Y 327.989,Z 614.475,A -85,B 0,C 180,E1 2918.424,E2 2918.424} C_VEL
LIN {X 0,Y 324.29,Z 611.139,A -85,B 0,C 180,E1 2914.67,E2 2914.67} C_VEL
LIN {X 0,Y 321.825,Z 608.69,A -85,B 0,C 180,E1 2912.302,E2 2912.302} C_VEL
LIN {X 0,Y 317.681,Z 605.829,A -85,B 0,C 180,E1 2908.786,E2 2908.786} C_VEL
LIN {X 0,Y 313.258,Z 602.076,A -85,B 0,C 180,E1 2905.322,E2 2905.322} C_VEL
LIN {X 0,Y 310.416,Z 600.177,A -85,B 0,C 180,E1 2903.34,E2 2903.34} C_VEL
LIN {X 0,Y 305.05,Z 596.732,A -85,B 0,C 180,E1 2899.93,E2 2899.93} C_VEL
LIN {X 0,Y 297.426,Z 589.942,A -85,B 0,C 180,E1 2894.404,E2 2894.404} C_VEL
LIN {X 0,Y 293.182,Z 583.796,A -85,B 0,C 180,E1 2889.62,E2 2889.62} C_VEL
LIN {X 0,Y 291.211,Z 577.996,A -85,B 0,C 180,E1 2885.489,E2 2885.489} C_VEL
LIN {X 0,Y 287.233,Z 603.015,A -85,B 0,C 180,E1 2885.22,E2 2885.22} C_VEL
LIN {X 0,Y 281.631,Z 626.103,A -85,B 0,C 180,E1 2884.996,E2 2884.996} C_VEL
LIN {X 0,Y 274.404,Z 648.012,A -85,B 0,C 180,E1 2884.771,E2 2884.771} C_VEL
LIN {X 0,Y 265.767,Z 668.568,A -85,B 0,C 180,E1 2884.48,E2 2884.48} C_VEL
LIN {X 0,Y 254.593,Z 690.255,A -85,B 0,C 180,E1 2884.05,E2 2884.05} C_VEL
LIN {X 0,Y 242.415,Z 709.853,A -85,B 0,C 180,E1 2883.514,E2 2883.514} C_VEL
LIN {X 0,Y 228.234,Z 729.054,A -85,B 0,C 180,E1 2882.802,E2 2882.802} C_VEL
LIN {X 0,Y 214.09,Z 745.494,A -85,B 0,C 180,E1 2881.97,E2 2881.97} C_VEL
LIN {X 0,Y 197.988,Z 761.68,A -85,B 0,C 180,E1 2880.856,E2 2880.856} C_VEL
LIN {X 0,Y 180.978,Z 776.305,A -85,B 0,C 180,E1 2879.43,E2 2879.43} C_VEL
LIN {X 0,Y 162.756,Z 789.927,A -85,B 0,C 180,E1 2877.535,E2 2877.535} C_VEL
LIN {X 0,Y 143.529,Z 802.159,A -85,B 0,C 180,E1 2874.967,E2 2874.967} C_VEL
LIN {X 0,Y 125.284,Z 812.143,A -85,B 0,C 180,E1 2871.722,E2 2871.722} C_VEL
LIN {X 0,Y 104.84,Z 821.588,A -85,B 0,C 180,E1 2866.592,E2 2866.592} C_VEL
LIN {X 0,Y 85.597,Z 829.05,A -85,B 0,C 180,E1 2859.139,E2 2859.139} C_VEL
LIN {X 0,Y 67.777,Z 834.771,A -85,B 0,C 180,E1 2847.23,E2 2847.23} C_VEL
LIN {X 0,Y 55.244,Z 838.326,A -85,B 0,C 180,E1 2830.658,E2 2830.658} C_VEL
LIN {X 0,Y 48.539,Z 840.399,A -85,B 0,C 180,E1 2806.761,E2 2806.761} C_VEL
LIN {X 0,Y 48.061,Z 840.788,A -85,B 0,C 180,E1 2791.192,E2 2791.192} C_VEL
LIN {X 0,Y 48.172,Z 840.526,A -85,B 0,C 180,E1 2778.021,E2 2778.021} C_VEL
LIN {X 0,Y 52.655,Z 839.105,A -85,B 0,C 180,E1 2755.274,E2 2755.274} C_VEL
LIN {X 0,Y 64.384,Z 835.761,A -85,B 0,C 180,E1 2736.146,E2 2736.146} C_VEL
LIN {X 0,Y 81.06,Z 830.61,A -85,B 0,C 180,E1 2723.248,E2 2723.248} C_VEL
LIN {X 0,Y 100.338,Z 823.449,A -85,B 0,C 180,E1 2714.857,E2 2714.857} C_VEL
LIN {X 0,Y 117.747,Z 815.804,A -85,B 0,C 180,E1 2709.939,E2 2709.939} C_VEL
LIN {X 0,Y 137.723,Z 805.529,A -85,B 0,C 180,E1 2705.967,E2 2705.967} C_VEL
LIN {X 0,Y 156.226,Z 794.285,A -85,B 0,C 180,E1 2703.258,E2 2703.258} C_VEL
LIN {X 0,Y 175.005,Z 781.04,A -85,B 0,C 180,E1 2701.143,E2 2701.143} C_VEL
LIN {X 0,Y 191.972,Z 767.049,A -85,B 0,C 180,E1 2699.614,E2 2699.614} C_VEL
LIN {X 0,Y 208.043,Z 751.874,A -85,B 0,C 180,E1 2698.424,E2 2698.424} C_VEL
LIN {X 0,Y 210.18,Z 749.648,A -85,B 0,C 180,E1 2698.284,E2 2698.284} C_VEL
LIN {X 0,Y 215.31,Z 744.241,A -85,B 0,C 180,E1 2697.69,E2 2697.69} C_VEL
LIN {X 0,Y 227.406,Z 730.61,A -85,B 0,C 180,E1 2695.478,E2 2695.478} C_VEL
LIN {X 0,Y 232.066,Z 724.701,A -85,B 0,C 180,E1 2695.017,E2 2695.017} C_VEL
LIN {X 0,Y 245.391,Z 706.105,A -85,B 0,C 180,E1 2694.486,E2 2694.486} C_VEL
LIN {X 0,Y 257.334,Z 686.427,A -85,B 0,C 180,E1 2694.07,E2 2694.07} C_VEL
LIN {X 0,Y 267.539,Z 666.105,A -85,B 0,C 180,E1 2693.761,E2 2693.761} C_VEL
LIN {X 0,Y 276.209,Z 644.94,A -85,B 0,C 180,E1 2693.535,E2 2693.535} C_VEL
LIN {X 0,Y 283.323,Z 622.648,A -85,B 0,C 180,E1 2693.357,E2 2693.357} C_VEL
LIN {X 0,Y 288.599,Z 600.149,A -85,B 0,C 180,E1 2693.165,E2 2693.165} C_VEL
LIN {X 0,Y 290.615,Z 588.154,A -85,B 0,C 180,E1 2693.034,E2 2693.034} C_VEL
LIN {X 0,Y 294.477,Z 596.187,A -85,B 0,C 180,E1 2687.15,E2 2687.15} C_VEL
LIN {X 0,Y 299.148,Z 601.067,A -85,B 0,C 180,E1 2682.995,E2 2682.995} C_VEL
LIN {X 0,Y 306.44,Z 606.677,A -85,B 0,C 180,E1 2678.163,E2 2678.163} C_VEL
LIN {X 0,Y 311.027,Z 609.488,A -85,B 0,C 180,E1 2675.094,E2 2675.094} C_VEL
LIN {X 0,Y 315.546,Z 613.334,A -85,B 0,C 180,E1 2671.621,E2 2671.621} C_VEL
LIN {X 0,Y 320.044,Z 616.418,A -85,B 0,C 180,E1 2667.92,E2 2667.92} C_VEL
LIN {X 0,Y 322.65,Z 618.895,A -85,B 0,C 180,E1 2665.516,E2 2665.516} C_VEL
LIN {X 0,Y 326.464,Z 622.247,A -85,B 0,C 180,E1 2661.782,E2 2661.782} C_VEL
LIN {X 0,Y 330.321,Z 624.93,A -85,B 0,C 180,E1 2657.866,E2 2657.866} C_VEL
LIN {X 0,Y 333.464,Z 628.348,A -85,B 0,C 180,E1 2654.224,E2 2654.224} C_VEL
LIN {X 0,Y 336.364,Z 630.733,A -85,B 0,C 180,E1 2650.712,E2 2650.712} C_VEL
LIN {X 0,Y 339.322,Z 632.494,A -85,B 0,C 180,E1 2647.01,E2 2647.01} C_VEL
LIN {X 0,Y 341.82,Z 635.585,A -85,B 0,C 180,E1 2643.36,E2 2643.36} C_VEL
LIN {X 0,Y 344.225,Z 637.792,A -85,B 0,C 180,E1 2639.589,E2 2639.589} C_VEL
LIN {X 0,Y 346.297,Z 639.155,A -85,B 0,C 180,E1 2636.031,E2 2636.031} C_VEL
LIN {X 0,Y 348.312,Z 640.067,A -85,B 0,C 180,E1 2632.266,E2 2632.266} C_VEL
LIN {X 0,Y 349.278,Z 641.058,A -85,B 0,C 180,E1 2630.091,E2 2630.091} C_VEL
LIN {X 0,Y 350.633,Z 642.958,A -85,B 0,C 180,E1 2626.568,E2 2626.568} C_VEL
LIN {X 0,Y 351.692,Z 644.247,A -85,B 0,C 180,E1 2622.979,E2 2622.979} C_VEL
LIN {X 0,Y 352.645,Z 645.067,A -85,B 0,C 180,E1 2619.36,E2 2619.36} C_VEL
LIN {X 0,Y 353.161,Z 645.558,A -85,B 0,C 180,E1 2615.85,E2 2615.85} C_VEL
LIN {X 0,Y 353.558,Z 645.818,A -85,B 0,C 180,E1 2612.269,E2 2612.269} C_VEL
LIN {X 0,Y 353.526,Z 645.809,A -85,B 0,C 180,E1 2608.704,E2 2608.704} C_VEL
LIN {X 0,Y 353.351,Z 645.648,A -85,B 0,C 180,E1 2605.13,E2 2605.13} C_VEL
LIN {X 0,Y 352.752,Z 645.243,A -85,B 0,C 180,E1 2601.579,E2 2601.579} C_VEL
LIN {X 0,Y 351.966,Z 644.45,A -85,B 0,C 180,E1 2597.865,E2 2597.865} C_VEL
LIN {X 0,Y 350.903,Z 643.351,A -85,B 0,C 180,E1 2594.385,E2 2594.385} C_VEL
LIN {X 0,Y 349.559,Z 641.509,A -85,B 0,C 180,E1 2590.623,E2 2590.623} C_VEL
LIN {X 0,Y 348.487,Z 640.143,A -85,B 0,C 180,E1 2588.101,E2 2588.101} C_VEL
LIN {X 0,Y 346.649,Z 639.309,A -85,B 0,C 180,E1 2584.529,E2 2584.529} C_VEL
LIN {X 0,Y 344.478,Z 637.972,A -85,B 0,C 180,E1 2580.816,E2 2580.816} C_VEL
LIN {X 0,Y 342.043,Z 635.848,A -85,B 0,C 180,E1 2577.03,E2 2577.03} C_VEL
LIN {X 0,Y 339.639,Z 632.957,A -85,B 0,C 180,E1 2573.483,E2 2573.483} C_VEL
LIN {X 0,Y 338.39,Z 631.97,A -85,B 0,C 180,E1 2571.81,E2 2571.81} C_VEL
LIN {X 0,Y 335.28,Z 629.939,A -85,B 0,C 180,E1 2567.95,E2 2567.95} C_VEL
LIN {X 0,Y 332.328,Z 627.263,A -85,B 0,C 180,E1 2564.508,E2 2564.508} C_VEL
LIN {X 0,Y 329.632,Z 624.344,A -85,B 0,C 180,E1 2561.395,E2 2561.395} C_VEL
LIN {X 0,Y 325.93,Z 621.83,A -85,B 0,C 180,E1 2557.679,E2 2557.679} C_VEL
LIN {X 0,Y 322.154,Z 618.411,A -85,B 0,C 180,E1 2554.039,E2 2554.039} C_VEL
LIN {X 0,Y 320.027,Z 616.415,A -85,B 0,C 180,E1 2552.082,E2 2552.082} C_VEL
LIN {X 0,Y 315.774,Z 613.507,A -85,B 0,C 180,E1 2548.563,E2 2548.563} C_VEL
LIN {X 0,Y 311.225,Z 609.673,A -85,B 0,C 180,E1 2545.049,E2 2545.049} C_VEL
LIN {X 0,Y 307.275,Z 607.191,A -85,B 0,C 180,E1 2542.378,E2 2542.378} C_VEL
LIN {X 0,Y 301.043,Z 602.817,A -85,B 0,C 180,E1 2538.392,E2 2538.392} C_VEL
LIN {X 0,Y 295.903,Z 597.796,A -85,B 0,C 180,E1 2534.28,E2 2534.28} C_VEL
LIN {X 0,Y 291.886,Z 591.752,A -85,B 0,C 180,E1 2529.464,E2 2529.464} C_VEL
LIN {X 0,Y 290.667,Z 588.147,A -85,B 0,C 180,E1 2526.952,E2 2526.952} C_VEL
LIN {X 0,Y 286.047,Z 612.086,A -85,B 0,C 180,E1 2526.729,E2 2526.729} C_VEL
LIN {X 0,Y 279.782,Z 634.552,A -85,B 0,C 180,E1 2526.556,E2 2526.556} C_VEL
LIN {X 0,Y 272.133,Z 655.492,A -85,B 0,C 180,E1 2526.368,E2 2526.368} C_VEL
LIN {X 0,Y 262.438,Z 676.707,A -85,B 0,C 180,E1 2526.092,E2 2526.092} C_VEL
LIN {X 0,Y 251.719,Z 696.13,A -85,B 0,C 180,E1 2525.739,E2 2525.739} C_VEL
LIN {X 0,Y 238.458,Z 716.155,A -85,B 0,C 180,E1 2525.245,E2 2525.245} C_VEL
LIN {X 0,Y 225.212,Z 733.134,A -85,B 0,C 180,E1 2524.677,E2 2524.677} C_VEL
LIN {X 0,Y 209.444,Z 750.569,A -85,B 0,C 180,E1 2523.877,E2 2523.877} C_VEL
LIN {X 0,Y 193.215,Z 765.905,A -85,B 0,C 180,E1 2522.9,E2 2522.9} C_VEL
LIN {X 0,Y 175.989,Z 780.079,A -85,B 0,C 180,E1 2521.628,E2 2521.628} C_VEL
LIN {X 0,Y 156.974,Z 793.392,A -85,B 0,C 180,E1 2519.876,E2 2519.876} C_VEL
LIN {X 0,Y 138.096,Z 804.717,A -85,B 0,C 180,E1 2517.613,E2 2517.613} C_VEL
LIN {X 0,Y 117.569,Z 815.108,A -85,B 0,C 180,E1 2514.264,E2 2514.264} C_VEL
LIN {X 0,Y 99.472,Z 822.821,A -85,B 0,C 180,E1 2510.075,E2 2510.075} C_VEL
LIN {X 0,Y 79.476,Z 829.929,A -85,B 0,C 180,E1 2502.959,E2 2502.959} C_VEL
LIN {X 0,Y 61.382,Z 835.111,A -85,B 0,C 180,E1 2491.592,E2 2491.592} C_VEL
LIN {X 0,Y 47.66,Z 838.473,A -85,B 0,C 180,E1 2473.811,E2 2473.811} C_VEL
LIN {X 0,Y 40.522,Z 840.212,A -85,B 0,C 180,E1 2447.223,E2 2447.223} C_VEL
LIN {X 0,Y 40.081,Z 840.558,A -85,B 0,C 180,E1 2430,E2 2430} C_VEL
LIN {X 0,Y 40.666,Z 840.18,A -85,B 0,C 180,E1 2411.36,E2 2411.36} C_VEL
LIN {X 0,Y 48.74,Z 838.213,A -85,B 0,C 180,E1 2384.113,E2 2384.113} C_VEL
LIN {X 0,Y 62.908,Z 834.715,A -85,B 0,C 180,E1 2367.122,E2 2367.122} C_VEL
LIN {X 0,Y 82.119,Z 829.083,A -85,B 0,C 180,E1 2355.877,E2 2355.877} C_VEL
LIN {X 0,Y 102.29,Z 821.705,A -85,B 0,C 180,E1 2349.168,E2 2349.168} C_VEL
LIN {X 0,Y 122.415,Z 812.879,A -85,B 0,C 180,E1 2344.838,E2 2344.838} C_VEL
LIN {X 0,Y 142.051,Z 802.473,A -85,B 0,C 180,E1 2341.859,E2 2341.859} C_VEL
LIN {X 0,Y 161.736,Z 790.26,A -85,B 0,C 180,E1 2339.646,E2 2339.646} C_VEL
LIN {X 0,Y 180.074,Z 776.854,A -85,B 0,C 180,E1 2338.046,E2 2338.046} C_VEL
LIN {X 0,Y 197.267,Z 762.332,A -85,B 0,C 180,E1 2336.838,E2 2336.838} C_VEL
LIN {X 0,Y 214.018,Z 745.796,A -85,B 0,C 180,E1 2335.876,E2 2335.876} C_VEL
LIN {X 0,Y 228.268,Z 729.423,A -85,B 0,C 180,E1 2335.183,E2 2335.183} C_VEL
LIN {X 0,Y 232.066,Z 724.701,A -85,B 0,C 180,E1 2335.017,E2 2335.017} C_VEL
LIN {X 0,Y 236.617,Z 718.737,A -85,B 0,C 180,E1 2334.581,E2 2334.581} C_VEL
LIN {X 0,Y 247.634,Z 703.698,A -85,B 0,C 180,E1 2332.794,E2 2332.794} C_VEL
LIN {X 0,Y 251.814,Z 697.259,A -85,B 0,C 180,E1 2332.457,E2 2332.457} C_VEL
LIN {X 0,Y 262.393,Z 678.438,A -85,B 0,C 180,E1 2332.185,E2 2332.185} C_VEL
LIN {X 0,Y 272.114,Z 657.751,A -85,B 0,C 180,E1 2331.974,E2 2331.974} C_VEL
LIN {X 0,Y 280.046,Z 636.658,A -85,B 0,C 180,E1 2331.829,E2 2331.829} C_VEL
LIN {X 0,Y 286.551,Z 614.091,A -85,B 0,C 180,E1 2331.694,E2 2331.694} C_VEL
LIN {X 0,Y 289.974,Z 598.447,A -85,B 0,C 180,E1 2331.535,E2 2331.535} C_VEL
LIN {X 0,Y 293.319,Z 604.677,A -85,B 0,C 180,E1 2326.698,E2 2326.698} C_VEL
LIN {X 0,Y 297.179,Z 608.773,A -85,B 0,C 180,E1 2323.181,E2 2323.181} C_VEL
LIN {X 0,Y 304.742,Z 614.614,A -85,B 0,C 180,E1 2318.035,E2 2318.035} C_VEL
LIN {X 0,Y 309.095,Z 617.326,A -85,B 0,C 180,E1 2315.132,E2 2315.132} C_VEL
LIN {X 0,Y 313.921,Z 621.325,A -85,B 0,C 180,E1 2311.461,E2 2311.461} C_VEL
LIN {X 0,Y 318.524,Z 624.366,A -85,B 0,C 180,E1 2307.749,E2 2307.749} C_VEL
LIN {X 0,Y 322.645,Z 628.345,A -85,B 0,C 180,E1 2303.928,E2 2303.928} C_VEL
LIN {X 0,Y 326.553,Z 631.267,A -85,B 0,C 180,E1 2300.214,E2 2300.214} C_VEL
LIN {X 0,Y 328.953,Z 632.971,A -85,B 0,C 180,E1 2297.799,E2 2297.799} C_VEL
LIN {X 0,Y 332.322,Z 636.456,A -85,B 0,C 180,E1 2294.022,E2 2294.022} C_VEL
LIN {X 0,Y 335.552,Z 638.901,A -85,B 0,C 180,E1 2290.285,E2 2290.285} C_VEL
LIN {X 0,Y 338.374,Z 640.701,A -85,B 0,C 180,E1 2286.796,E2 2286.796} C_VEL
LIN {X 0,Y 340.942,Z 643.759,A -85,B 0,C 180,E1 2283.056,E2 2283.056} C_VEL
LIN {X 0,Y 343.485,Z 645.932,A -85,B 0,C 180,E1 2279.159,E2 2279.159} C_VEL
LIN {X 0,Y 345.751,Z 647.291,A -85,B 0,C 180,E1 2275.339,E2 2275.339} C_VEL
LIN {X 0,Y 347.605,Z 648.12,A -85,B 0,C 180,E1 2271.708,E2 2271.708} C_VEL
LIN {X 0,Y 349.103,Z 650.189,A -85,B 0,C 180,E1 2268.018,E2 2268.018} C_VEL
LIN {X 0,Y 350.223,Z 651.608,A -85,B 0,C 180,E1 2264.719,E2 2264.719} C_VEL
LIN {X 0,Y 351.26,Z 652.727,A -85,B 0,C 180,E1 2260.877,E2 2260.877} C_VEL
LIN {X 0,Y 352.027,Z 653.312,A -85,B 0,C 180,E1 2257.343,E2 2257.343} C_VEL
LIN {X 0,Y 352.412,Z 653.669,A -85,B 0,C 180,E1 2253.741,E2 2253.741} C_VEL
LIN {X 0,Y 352.614,Z 653.784,A -85,B 0,C 180,E1 2250.325,E2 2250.325} C_VEL
LIN {X 0,Y 352.458,Z 653.675,A -85,B 0,C 180,E1 2246.748,E2 2246.748} C_VEL
LIN {X 0,Y 352.113,Z 653.442,A -85,B 0,C 180,E1 2243.478,E2 2243.478} C_VEL
LIN {X 0,Y 351.39,Z 652.83,A -85,B 0,C 180,E1 2239.673,E2 2239.673} C_VEL
LIN {X 0,Y 350.516,Z 651.93,A -85,B 0,C 180,E1 2236.137,E2 2236.137} C_VEL
LIN {X 0,Y 349.34,Z 650.543,A -85,B 0,C 180,E1 2232.683,E2 2232.683} C_VEL
LIN {X 0,Y 348.046,Z 648.516,A -85,B 0,C 180,E1 2229.132,E2 2229.132} C_VEL
LIN {X 0,Y 346.225,Z 647.551,A -85,B 0,C 180,E1 2225.609,E2 2225.609} C_VEL
LIN {X 0,Y 344.116,Z 646.363,A -85,B 0,C 180,E1 2221.921,E2 2221.921} C_VEL
LIN {X 0,Y 341.828,Z 644.55,A -85,B 0,C 180,E1 2218.231,E2 2218.231} C_VEL
LIN {X 0,Y 339.287,Z 641.886,A -85,B 0,C 180,E1 2214.512,E2 2214.512} C_VEL
LIN {X 0,Y 337.573,Z 640.047,A -85,B 0,C 180,E1 2212.186,E2 2212.186} C_VEL
LIN {X 0,Y 334.592,Z 638.267,A -85,B 0,C 180,E1 2208.595,E2 2208.595} C_VEL
LIN {X 0,Y 331.202,Z 635.387,A -85,B 0,C 180,E1 2204.7,E2 2204.7} C_VEL
LIN {X 0,Y 327.946,Z 632.093,A -85,B 0,C 180,E1 2201.145,E2 2201.145} C_VEL
LIN {X 0,Y 324.091,Z 629.512,A -85,B 0,C 180,E1 2197.428,E2 2197.428} C_VEL
